# B&R Automation Studio project TD52 (part 27)

#### EleStartCyclic.st
```iecst
 (********************************************************************
EleStart		engine start/stop control: electrical starter equipment

This code is confidential and proprietary to the INNIO Company.
It may not be used in any form, or reproduced in any manner,
without the express written permission of the INNIO Company.
Copyright, INNIO Company, 2025

Customized modifications: -
------------------------

History:
-------
V01		10.07.1998 Pa			erstellt
V2.20.3	30.11.2007 LH			Ausspuren Starter bei Zahn auf Zahn
V2.30.0	16.01.2008 LH			Blockierung Modul angepasst für Insel nach Ablauf KU-Filter
 		30.01.2008 LH			Ansteuerung MEGA-Gasventile
 		02.04.2008 LH			1-maliges Absetzen von UW-EIN nach Kaltstart
V2.33.0	17.07.2008 lettenb.		sel_GlowIgnPrevent added
V2.34.0	22.10.2008 lettenb.		AT4_BLOCK added, block.ack.by starter temp.(op.message 3300)
								bs_15s_rel_oper added
		03.12.2008 lettenb.		ZM_GASV: M_GASV added
V2.50.0	28.01.2009 lettenb.		ZM_M_BLOCK: M_ST_VORW removed
			   	            	puff_mini removed
		06.04.2009 lett./gföll./plattner	Vorschmierzeit fix mit 60 = ersatz für TW_T85
								überbrückung T_VERZ_ANF bei notstrom(M_NANF)
V2.60.0	07.08.2009 lettenb.		udp_dmnd, udp_comm removed, ANF_NB added
								ssExtPwrSetP1, ssExtPwrSetP2, DI_ExtPwrSetP1, DI_ExtPwrSetP2 added
								custom.counter1-4 moved to c_amm
V3.10.0	19.01.2010 lettenb.		QUITT_TUEV reset pulse according EN ISO 13849-1 / 5.2.2
								(d.h. Ausgangsimpuls an UW_EIN erst wenn der RESET-Taster losgelassen wird)
V3.20.0	05.08.2010 lettenb.		ton_RESET_4 added reset counter for AT4_BLOCK after cool down
		15.09.2010 MM (BuR)  	STARTER_IgnST included
		30.09.2010 MM (BuR)  	GS_EIN replaced with GCB_ON
		30.09.2010 MM(BuR) 		NW20 deleted (GCB_ON --> GCB_ON)
		30.09.2010 MM(BuR) 		M_GSEIN replaced with GCB_ON
		21.10.2010 lettenb. 	AW_EXPSH, AW_EXPSB, B_P_SOLL, B_P_RED, AW_EXDSH, AW_EXDSB, B_N_SOLL
								sel.ext.power setpoint moved to task: p_limits
		05.11.2010 lettenb.		purgecycle added
		07.12.2010 lettenb.		BLOCK_EVU added, ZUEND: contact STARTER_IgnST changed
		14.02.2011 lettenb.		selection duration start puls time added
V3.90.0	29.10.2012 lettenb.		logic for manual start prozedure changed
V3.99.0	14.02.2013 lettenb.		IN_AG.bGasMix_Ref(M_GM_Ref) removed, not supported from MM gas mixer
V3.99   28.02.2013 pankajrodey	Generated for modular software with changes for V3.30
V3.99.1	20.01.2014 lettenb.		man.start time 30" added
V3.99.2	05.12.2013 zengerer		ADAPTIVE maximum start time 22" to 35" with rTiFactor_Cylinders AND rTiFactor_Cylinders FOR series 4 deflagration, new OUT: bRel_Gasvalve for MM op_state
V3.99.3	09.12.2013 zengerer		CleanUp
V3.99.4	02.01.2014 zengerer		prepared FOR PILOT ENGINES: save statistic data of 200 starts in task Perm_AG
V3.99.5	29.01.2014 zengerer		bGV_Start_ScaveBlock, MM2VIS.rN_EngStart (and others) optional reactivated
V3.99.6	19.03.2014 zengerer		entered Para.bVISA to prevent use of new adoptive start, if VISA reglementation is selected
V4.00.1 09.05.2014 lettenb.		xEngType.Type4: OUT_AG.tChargeOff_Dem.Do added, bugfix
V4.00.1 19.05.2014 Denk			xTON_StartErr Startzeit von 20s --> 12s
V4.00.2 30.05.2014 lettenb.		startup failure counter also for man.starts, bugfix + cleanup
V4.00.3 30.06.2014 lettenb.		xEngType.Type2 added, bugfix
V4.00.4 01.10.2014 lettenb.		bugfix startup failure in combination with EG_Scav(BR3,4)
		03.11.2014				start duration times BR3,6 corr., bugfix
V4.00.5	03.02.2015				920 added
		20.04.2015				xTP_StarterON: phantomstart resolved
V4.04.0	18.11.2016				xTON_DelayStart.PT, xTON_DelayManStart.PT: 6->0s start delay removed(fahringer)
		21.12.2016 Denk			Modification for WinMOD simulation
V4.05.0	07.08.2017 Messner		Starter battery voltage monitoring
		01.02.2018 lettenb.		tiStarterOFF; define value at plc startup(when xCTD_Start.CV=0), bugfix(1st start too long/perktold)
V4.05.1	14.02.2018 Weitzerr		move starter battery voltage monitoring to task AuxGnl
		19.09.2018 lettenb.		switching off battery charge for BR2+3 identical to BR4(HW solution not working), bu
V4.06.0	19.09.2018 Perktold,	integrated OUT_AG.iStartCount
V4.07.0	25.10.2018 Schmid		xTON_RESET_4: only triggered with IN_AG.bEng_SU_Man, bugfix
V4.10.0	28.01.2021 Schmid		interface for ChargeOff_Dem for starter battery test added
		29.01.2021 Schmid		manual start stop buttons from Opstate instead of VIS
V4.12.0 21.12.2022 Bacci		Starter battery monitoring parameters added: Para.rN_StarterMonTtT_LimLo and Para.tiStarterMonDuration. W9074 added
		20.01.2023 Zengerer		Type3 flush start time preparation optional with bOptType3AdoptiveStartEnab
V4.13.0	21.07.2023 Bacci		Type3 new starting procedure and adaptive first start attempt (bOptType3AdoptiveStartEnab deleted)
		20.11.2023 Bacci		Starter/s correct engagement monitoring added
V4.14.0	25.11.2024 Bacci		T6 Start procedure with purge start (2024-219)
V4.25.0	10.09.2025 Bacci	 	Include purge air calculation via SafetyPLC (2025-260)

Instructions for use:
--------------------
Outstandings:
------------
(*********************************************************************)

PROGRAM _CYCLIC

	(* Engine Type 9 - Return *)
	IF xEngType.Type9 THEN RETURN;
    END_IF;

	IF xEngType.Type6 THEN
		xR_TRIG_bParaSetupOk(CLK := IN_AG.tPB2MM.bParaSetupOk);
		IF xR_TRIG_bParaSetupOk.Q THEN
			rTi_ST_Active_zero := LIMIT(0, TIME_TO_REAL(Para.tiST_MaxDur_OverheatPrev)/1000 * (1 - (LIMIT(0.2, Para.rST_ReqOpTiAftCooldown, 1))), MAX(0,TIME_TO_REAL(Para.tiST_MaxDur_OverheatPrev)/1000));
		END_IF;
	ELSE
		rTi_ST_Active_zero := 0;
	END_IF;

	bAdoptiveStartEnab := (xEngType.Type4 OR xEngType.Type3) AND NOT Para.bVISA;

	IF xEngType.Type6 THEN							(* BR6 *)(* No longer used (2024-219) *)
		tiStarterON1 :=	 T#25s; 	(* = Total start time incl. flush cranking time at 1st start attempt in automatic *)
		tiStarterON2 :=	 T#20s;		(* = Total start time incl. flush cranking time at 2nd start attempt in automatic *)
		tiStarterON3 :=	 T#20s; 	(* = Total start time incl. flush cranking time at 3rd start attempt in automatic *)
		tiStartScav1 :=	 T#2s;		(* = flush cranking time wthout gas, for 1st start attempt *)
		tiStartScav2 :=	 T#2s;  	(* = flush cranking time wthout gas, for 2nd start attempt *)
		tiStartScav3 :=	 T#2s;  	(* = flush cranking time wthout gas, for 3rd start attempt *)
		tiStarterOFF1 := T#14s; 	(* = N.C. not in use *)
		tiStarterOFF2 := T#14s; 	(* = delay time until 2nd start attempt *)
		tiStarterOFF3 := T#14s; 	(* = delay time until 3rd start attempt *)
	ELSIF xEngType.Type4 AND NOT Para.bVISA THEN 	(* BR4 *)
		tiStarterON1 :=	 T#22s;		(* = Total start time incl. flush cranking time, base time for 1st start attempt- ADAPTIVE maximum time 22" (max.35" *)
		tiStarterON2 :=	 T#30s;		(* = Total start time incl. flush cranking time, for 2nd start attempt *)
		tiStarterON3 :=	 T#30s;		(* = Total start time incl. flush cranking time, for 3rd start attempt *)
		tiStartScav1 :=	 T#0s;		(* = flush cranking time wthout gas, for 1st start attempt- ADAPTIVE maximum time 22" to 35" *)
		tiStartScav2 :=	 T#10s;		(* = flush cranking time wthout gas, for 2nd start attempt *)
		tiStartScav3 :=	 T#10s;		(* = flush cranking time wthout gas, for 3rd start attempt *)
		tiStarterOFF1 := T#15s;		(* = n.c. *)
		tiStarterOFF2 := T#12s;		(* = delay time until 2nd start attempt *)
		tiStarterOFF3 := T#301s;	(* = delay time until 3rd start attempt *)
	ELSIF xEngType.Type3 AND NOT Para.bVISA THEN 		(* BR3 option with flush hardware *)
		tiStarterON1 :=	 T#34s;		(* = Total start time incl. flush cranking time, base time for 1st start attempt- ADAPTIVE maximum time 34" (max.40" *)
		tiStarterON2 :=	 T#30s;		(* = Total starg time incl. flush cranking time, time for 2nd start attempt *)
		tiStarterON3 :=	 T#30s;		(* = Total start time incl. flush cranking time, time for 3rd start attempt *)
		tiStartScav1 :=	 T#10s;		(* = flush cranking time wthout gas, for 1st start attempt- ADAPTIVE maximum time 22" to 35" *)
		tiStartScav2 :=	 T#10s;		(* = flush cranking time wthout gas, for 2nd start attempt *)
		tiStartScav3 :=	 T#10s;		(* = flush cranking time wthout gas, for 3rd start attempt *)
		tiStarterOFF1 := T#15s;		(* = n.c. *)
		tiStarterOFF2 := T#12s;		(* = delay time until 2nd start attempt *)
		tiStarterOFF3 := T#301s;	(* = delay time until 3rd start attempt *)
	ELSE											(* BR2,BR3 with standard hardware *)
		tiStarterON1 :=	 T#20s; 	(* = Total start time incl. flush cranking time, for 1st start attempt *)
		tiStarterON2 :=	 T#20s;		(* = Total start time incl. flush cranking time, for 2nd start attempt *)
		tiStarterON3 :=	 T#20s;		(* = Total start time incl. flush cranking time, for 3rd start attempt *)
		tiStartScav1 :=	 T#0s;		(* = flush cranking time wthout gas, for 1st start attempt *)
		tiStartScav2 :=	 T#0s;		(* = flush cranking time wthout gas, for 2nd start attempt *)
		tiStartScav3 :=	 T#0s;		(* = flush cranking time wthout gas, for 3rd start attempt *)
		tiStarterOFF1 := T#12s;		(* = n.c. *)
		tiStarterOFF2 := T#12s;		(* = delay time until 2nd start attempt *)
		tiStarterOFF3 := T#12s;		(* = delay time until 3rd start attempt *)
	END_IF;

	IF rTiFactor_Cylinders = 0 THEN	rTiFactor_Cylinders := 0.99; END_IF;
	IF rTiFactor_N_EngStart= 0 THEN	rTiFactor_N_EngStart:= 0.99; END_IF;

	(* start stop button info from Opstate *)
	bStart 	:= IN_AG.bStart;
	bStop 	:= IN_AG.bStop;

	(* -------------------------------------------------------------------------------------------------------------------------------------- *)
	(* New type 6 starting procedure *)

	(* ------------------------------------------------------------------------------------ *)
	(* EleStart cycle time *)
	RTInfo_CTR(enable := TRUE);
	tiCycleTime := UDINT_TO_TIME(RTInfo_CTR.cycle_time)/1000;		// time variable
	rCycleTime := UDINT_TO_REAL(RTInfo_CTR.cycle_time)/1000000;  	// real variable in seconds

	(* ------------------------------------------------------------------------------------ *)
	(* Set parameter 15074 "Minimum air volume required for system purge" based on parameter 11303 "exhaust gas scavenging active" and EPS demand *)
	IF xEngType.Type6 THEN
		IF NOT Para.bEGScav_Active THEN 				// Exhaust gas scavenging not active
			IF xEngType.Motortype = 612 THEN
				IF IN_AG.bEng_Dem_EPS THEN
					iVol_MinAirLim_SysPurge := 680;
				ELSE
					iVol_MinAirLim_SysPurge := MAX(680, Para.iVol_MinAir_SysPurge);
				END_IF;
			ELSIF xEngType.Motortype = 616 THEN
				IF IN_AG.bEng_Dem_EPS THEN
					iVol_MinAirLim_SysPurge := 750;
				ELSE
					iVol_MinAirLim_SysPurge := MAX(750, Para.iVol_MinAir_SysPurge);
				END_IF;
			ELSIF xEngType.Motortype = 620 THEN
				IF IN_AG.bEng_Dem_EPS THEN
					iVol_MinAirLim_SysPurge := 800;
				ELSE
					iVol_MinAirLim_SysPurge := MAX(800, Para.iVol_MinAir_SysPurge);
				END_IF;
			ELSIF xEngType.Motortype = 624 THEN
				IF IN_AG.bEng_Dem_EPS THEN
					iVol_MinAirLim_SysPurge := 1400;
				ELSE
					iVol_MinAirLim_SysPurge := MAX(1400, Para.iVol_MinAir_SysPurge);
				END_IF;
			END_IF;
		ELSIF Para.bEGScav_Active AND (IN_AG.bEng_Dem_EPS AND (NOT Para.bEGScav_ifAuxV_ok OR NOT IN_AG.tAuxV_Eng_ok.Di)) THEN 				// Exhaust gas scavenging active, but not executed during EPS
			IF xEngType.Motortype = 612 THEN
				iVol_MinAirLim_SysPurge := 680;
			ELSIF xEngType.Motortype = 616 THEN
				iVol_MinAirLim_SysPurge := 750;
			ELSIF xEngType.Motortype = 620 THEN
				iVol_MinAirLim_SysPurge := 800;
			ELSIF xEngType.Motortype = 624 THEN
				iVol_MinAirLim_SysPurge := 1400;
			END_IF;
		ELSE
			iVol_MinAirLim_SysPurge := 0;
		END_IF;
	ELSE
		iVol_MinAirLim_SysPurge := 0;
	END_IF;

	(* ------------------------------------------------------------------------------------ *)
	(* Volume flow through the engine *)
	IF xEngType.Type6 THEN
		rVol_CylDis :=	((UINT_TO_REAL(xEngType.Bore)/1000/2) ** 2 * brmPI * UINT_TO_REAL(xEngType.Stroke)/1000) * 1000; 								// single cylinder displacement [lt], //	Volume [lt]	:=	(( radius [m] ) ^ 2 * PI * ( stroke [m] ))*1000
		IF IN_AG.rN_EngAct > 50 THEN
			rVolFlow_RunEng := LIMIT(0, Para.rVolEff_CrkSpeed * rVol_CylDis * UINT_TO_REAL(xEngType.NumberOfCylinder) * IN_AG.rN_EngAct/120, 20000);	// volume flow through the engine REAL [lt/s]
		ELSE
			rVolFlow_RunEng := 0;
		END_IF;
		iVolFlow_RunEng := REAL_TO_UDINT(rVolFlow_RunEng);																								// volume flow through the engine UDINT [lt/s]
	ELSE
		rVol_CylDis := 0;
		rVolFlow_RunEng := 0;
		iVolFlow_RunEng := 0;
	END_IF;

	(* ------------------------------------------------------------------------------------ *)
	(* Volume of mixture calculation *)
	xTON_GVOpen_1s(IN:= IN_AG.bGV_On, PT:= T#1s);																								// gas valve open for more than 1 second

	IF xEngType.Type6 THEN
		//Fuel admition status
		IF xTON_GVOpen_1s.Q  THEN
			 rFuelAdm := 1;
		ELSE
			 rFuelAdm := (Para.rVolFlow_Marg - 1);
		END_IF;

		IF IN_AG.rN_EngAct = 0 OR OUT_AG.tEleStarter_Dem.Do THEN 																				// during engine standstill and during cranking phase
			rVol_Mx := LIMIT(0, rVol_Mx + rFuelAdm * rVolFlow_RunEng * rCycleTime, LIMIT(100, UDINT_TO_REAL(Para.iVol_TolUnbrtMxMax), 5000));
		ELSIF IN_AG.rN_EngAct <> 0 AND NOT IN_AG.bGV_On AND NOT OUT_AG.tEleStarter_Dem.Do  THEN													// during shut down phase
			rVol_Mx := LIMIT(0, rVol_Mx + rFuelAdm * rVolFlow_RunEng * rCycleTime, UDINT_TO_REAL(Para.iVol_PremxInSys));
		ELSIF M_DREHZ AND IN_AG.bGV_On THEN 																									// during engine operation
			rVol_Mx := UDINT_TO_REAL(Para.iVol_PremxInSys);
		END_IF;
	ELSE
		rFuelAdm := 0;
		rVol_Mx := 0;
	END_IF;

	(* ------------------------------------------------------------------------------------ *)
	(* Purge state identification *)
	IF xEngType.Type6 THEN
		(* Volume of purge air calculation *)
		IF IN_AG.bSafetyPLC_Active AND NOT Para.bEGScav_Active THEN 														//coming from safety PLC 	(* SAFETY PLC *)
			rVol_PurgeAir := IN_AG.rVol_PurgeAir_SafeOUT;																								(* SAFETY PLC *)
		ELSIF xTON_GVOpen_1s.Q OR bFail_PurgeCrk THEN																									(* SAFETY PLC *)
			rVol_PurgeAir := 0;
		ELSE
			rVol_PurgeAir := LIMIT(0, rVol_PurgeAir + rVolFlow_RunEng * (1 - Para.rVolFlow_Marg) * rCycleTime, 100000);		// volume of purge air REAL [lt]
		END_IF;
		iVol_PurgeAir := REAL_TO_UDINT(rVol_PurgeAir);																		// volume of purge air UDINT [lt]

		(* Purge state *)
		(* detect reset of emergancy operation demand  *)
		xF_TRIG_bEng_Dem_EPS(CLK := IN_AG.bEng_Dem_EPS);
		IF xF_TRIG_bEng_Dem_EPS.Q THEN
			bSt_Purge := FALSE;																								// set purge status to false after emergency operation demand reset
		END_IF;

		IF IN_AG.bSafetyPLC_Active AND NOT Para.bEGScav_Active THEN 														//coming from safety PLC 	(* SAFETY PLC *)
			bSt_Purge := IN_AG.bSafeOUT_Purge_OK;																										(* SAFETY PLC *)
		ELSIF xTON_GVOpen_1s.Q THEN 																													(* SAFETY PLC *)
			bSt_Purge := FALSE;
		ELSIF (rVol_PurgeAir >= UDINT_TO_REAL(iVol_MinAirLim_SysPurge)) THEN
			bSt_Purge := TRUE;
		END_IF;

		(* detect successful purge cranking cycle *)
		xR_TRIG_bSt_Purge(CLK := bSt_Purge);
	ELSE
		rVol_PurgeAir := 0;
		iVol_PurgeAir := 0;
		bSt_Purge := FALSE;
	END_IF;

	(* ------------------------------------------------------------------------------------ *)
	(* Starter temperature monitoring *)
	IF xEngType.Type6 THEN
		(* detect beginning of starter cool down phase *)
		xF_TRIG_bEleStarter_Dem(CLK := OUT_AG.tEleStarter_Dem.Do);
		IF xF_TRIG_bEleStarter_Dem.Q THEN
			rTi_ST_Active_zero := rTi_ST_Active;
			rTi_ST_Cooldown := 0;
		END_IF;

		(* Cumulated starting time calculation REAL [s] *)
		IF OUT_AG.tEleStarter_Dem.Do THEN
			rTi_ST_Active := LIMIT(0, rTi_ST_Active + Para.rST_Heatup_Fact * rCycleTime, MAX(0,TIME_TO_REAL(Para.tiST_MaxDur_OverheatPrev)/1000));																// Starter in use, heat up phase
		ELSE
			rTi_ST_Active := LIMIT(0, rTi_ST_Active_zero * EXP(-(rTi_ST_Cooldown / LIMIT(100, TIME_TO_REAL(Para.tiST_CooldownConst)/1000, 9000))), MAX(0,TIME_TO_REAL(Para.tiST_MaxDur_OverheatPrev)/1000));	// Starter not in use, cool down phase
			rTi_ST_Cooldown := rTi_ST_Cooldown + rCycleTime;
		END_IF;

		IF rTi_ST_Active < 1 AND NOT OUT_AG.tEleStarter_Dem.Do THEN 				// Rounding for small values
			rTi_ST_Active := 0;
			rTi_ST_Cooldown := 0;
			rTi_ST_Active_zero := 0;
		END_IF;

		(* Calculation of remaining starting time [s] *)
		rTi_ST_Res := TIME_TO_REAL(Para.tiST_MaxDur_OverheatPrev)/1000 - rTi_ST_Active;
		iTi_ST_Res := REAL_TO_INT(rTi_ST_Res);

		(* Calculation of starter temperature status *)
		xGR_MINR_bSt_STT (In:= rTi_ST_Res, Gw:= 0, Hy:= LIMIT(0, TIME_TO_REAL(Para.tiST_MaxDur_OverheatPrev)/1000 * (LIMIT(0.2, Para.rST_ReqOpTiAftCooldown, 1)), MAX(0,(TIME_TO_REAL(Para.tiST_MaxDur_OverheatPrev)/1000)-1)));
		bSt_STT := NOT xGR_MINR_bSt_STT.Q;
	ELSE
		rTi_ST_Active_zero := 0;
		rTi_ST_Cooldown := 0;
		rTi_ST_Active := 0;
		rTi_ST_Res := 0;
		iTi_ST_Res := 0;
		bSt_STT := FALSE;
	END_IF;

	//note:
	//		1.	the division by zero in the exponential calculation has been prevented using the boundaries limits decided for Para.tiST_CooldownConst
	//		2.	The upper limit of xGR_MINR_bSt_STT is used to be able to set the starter temperature status to true when Para.rST_ReqOpTiAftCooldown is 100%.
	//			In such situation, since rTi_ST_Res is never higher than TIME_TO_REAL(Para.tiST_MaxDur_OverheatPrev)/1000,  xGR_MINR_bSt_STT would never go to FALSE
	//			The cumulated starting time is forced to 0 when it´s value is < than 1s. The same trashold has been used also on the remining starting time.
	//			When rTi_ST_Res is > maximunm starting duration - 1s  the starter temperature status is set to TRUE (xGR_MINR_bSt_STT goes to false)

	(* ------------------------------------------------------------------------------------ *)
	(* Manual request for purge cranking cycle and start attempt *)
	IF xEngType.Type6 THEN
		bEng_SU_Man_Req := 		(bStart OR bEng_SU_Man_Req)
								AND		 bOMSS_Man
								AND 	 IN_AG.bEng_Dem_Man
								AND 	(IN_AG.bEng_SU_Man OR bSt_RelAuxOff_STT)								// retain during waiting time for starter release
								AND(NOT IN_AG.bBlocDelay_ManStart OR OUT_AG.bEng_Start OR bSt_RelAuxOff_STT)
								AND     (IN_AG.bScavFinished OR NOT IN_AG.bRel_ScavN2)
								AND NOT (xR_TRIG_bSt_Purge.Q AND xCTD_Start.CV <> xCTD_Start.PV)				// reset request when the purge done and first start
								AND NOT xF_TRIG_bSt_RelAuxOff_STT.Q												// reset request when release form starter temperature is given
								AND NOT bStop;
	ELSE
		bEng_SU_Man_Req := FALSE;
	END_IF;

	(* ------------------------------------------------------------------------------------ *)
	(* fast start readiness from purge status and starter temperature capability *)
	IF xEngType.Type6 THEN
		OUT_AG.bFS_Rdy_STT_StPurge := ((rTi_ST_Res >= TIME_TO_REAL(Para.tiST_MaxDur_OverheatPrev)/1000 * (LIMIT(0.2, Para.rST_ReqOpTiAftCooldown, 1))) AND bSt_Purge);		// enough starter temperature capability and purge ok
	ELSE
		OUT_AG.bFS_Rdy_STT_StPurge := FALSE;
	END_IF;

	(* ------------------------------------------------------------------------------------ *)
	(* demand to open inlet louvers before purge cranking cycle for fast start *)
	IF xEngType.Type6 THEN
		bFS_Req	:= bOMSS_Aut AND IN_AG.bEng_Rel AND Para.bFSPreL_Act AND IN_AG.bPermPreLube_Dem;
		OUT_AG.bInLouDemAG := (bFS_Req AND OUT_AG.bPreL_FS_EngStaRel AND NOT IN_AG.bEng_Bloc) AND NOT M_DREHZ AND NOT (bSt_Purge OR bStartAtt_Run);
	ELSE
		bFS_Req := FALSE;
		OUT_AG.bInLouDemAG := FALSE;
	END_IF;

	(* ------------------------------------------------------------------------------------ *)
	(* Purge cranking cycle *)
	IF xEngType.Type6 THEN
		// Request purge cranking cycle
		bReq_PurgeCrk := (IN_AG.bEng_Dem_Aut AND NOT M_DREHZ AND (IN_AG.bEng_SU_Aut OR (bSt_RelAuxOff_STT AND bPurgeCrk_Run)) AND NOT (bSt_Purge OR bStartAtt_Run)) OR								// request during automatic start attempt
						 (IN_AG.bEng_Dem_Man AND NOT M_DREHZ AND bEng_SU_Man_Req AND (IN_AG.bEng_SU_Man OR (bSt_RelAuxOff_STT AND bPurgeCrk_Run)) AND NOT (bSt_Purge OR bStartAtt_Run)) OR		 	// request during manual start attempt
						 ((bFS_Req AND OUT_AG.bPreL_FS_EngStaRel AND NOT IN_AG.bEng_Bloc) AND NOT M_DREHZ AND NOT (bSt_Purge OR bStartAtt_Run) AND IN_AG.bInLouRelVE);								// request from fast start

		IF bReq_PurgeCrk THEN														// function activation
			bPurgeCrk_Run := TRUE;													// purge cranking cycle running
			bReq_Rel_STT_PurgeCrk := TRUE; 											// starter temperature release function requested from purge cranking cycle
			bGV_Block_PurgeCrk := TRUE; 											// GV blocked during purge cranking cycle
			bDem_ST_PurgeCrk := NOT bSt_RelAuxOff_STT; 								// starter demand from purge cranking
			IF bSpeedMon_PurgeCrkStartAtt THEN 										// purge cranking speed monitoring
				IF NOT bFail_StartAtt THEN
					bFail_PurgeCrk := TRUE;											// A2376 purge cranking cycle unsuccessful
				END_IF;
				bPurgeCrk_Run := FALSE;
				bReq_Rel_STT_PurgeCrk := FALSE;
				bGV_Block_PurgeCrk := FALSE;
				bDem_ST_PurgeCrk := FALSE;
			END_IF;
		ELSIF xR_TRIG_bSt_Purge.Q AND bEleStarter_Dem_PurgeCrk THEN  				// purge cranking cycle completed.
			bSfl_PurgeCrk := TRUE;													// B9088 purge cranking cycle successful
			bPurgeCrk_Run := FALSE;
			bReq_Rel_STT_PurgeCrk := FALSE;
			//bGV_Block_PurgeCrk := FALSE;											// for one extra cycle the starter is kept on and GV blocked
			//bDem_ST_PurgeCrk := FALSE;
			IF bSpeedMon_PurgeCrkStartAtt THEN 										// purge cranking speed monitoring active also during this cycle
				bFail_PurgeCrk := TRUE;												// A2376 purge cranking cycle unsuccessful
				bSfl_PurgeCrk := FALSE;
			END_IF;
		ELSE
			bPurgeCrk_Run := FALSE;
			bReq_Rel_STT_PurgeCrk := FALSE;
			bGV_Block_PurgeCrk := FALSE;
			bDem_ST_PurgeCrk := FALSE;
			bSfl_PurgeCrk := FALSE;
		END_IF;

		(* messages *)
		xTP_bSfl_PurgeCrk(IN := bSfl_PurgeCrk, PT:= T#5s);
		bMsg9097_set	:= bPurgeCrk_Run AND iVol_MinAirLim_SysPurge <> 0; 				// 9097 "purge cranking cycle initiated "
		bMsg2376_T6_set	:= bFail_PurgeCrk; 												// 2376 for T6 "Purge cranking cycle unsuccessful"
		bMsg9088_T6_set	:= xTP_bSfl_PurgeCrk.Q AND iVol_MinAirLim_SysPurge <> 0; 		// 9088 for T6 "Purge cranking cycle successful" active for 5s
	ELSE
		bReq_PurgeCrk := FALSE;
		bSfl_PurgeCrk := FALSE;
		bPurgeCrk_Run := FALSE;
		bReq_Rel_STT_PurgeCrk := FALSE;
		bGV_Block_PurgeCrk := FALSE;
		bDem_ST_PurgeCrk := FALSE;
		bFail_PurgeCrk := FALSE;
		xTP_bSfl_PurgeCrk(IN := FALSE, PT:= T#0s);
		bMsg9097_set := FALSE;
		bMsg2376_T6_set := FALSE;
		bMsg9088_T6_set := FALSE;
	END_IF;

	(* ------------------------------------------------------------------------------------ *)
	(* Start attempt*)
	IF xEngType.Type6 THEN
		// Request starter temperature release before engine start attempt
		xR_TRIG_bReq_Rel_STT_StartAtt(CLK := ((IN_AG.bEng_SU_Aut AND NOT M_DREHZ AND bSt_Purge AND NOT xCTD_Start.Q) OR
									 		  (IN_AG.bEng_SU_Man AND bEng_SU_Man_Req AND NOT M_DREHZ AND bSt_Purge AND NOT xCTD_Start.Q)));

		IF xR_TRIG_bReq_Rel_STT_StartAtt.Q THEN
			bRel_STT_StartAtt := FALSE;
		END_IF;

		bReq_StartAtt := (IN_AG.bEng_Dem_Aut AND NOT M_DREHZ AND (IN_AG.bEng_SU_Aut AND (bSt_Purge OR bStartAtt_Run)) AND bRel_STT_StartAtt AND NOT xCTD_Start.Q) OR
						 (IN_AG.bEng_Dem_Man AND NOT M_DREHZ AND bEng_SU_Man_Req AND (IN_AG.bEng_SU_Man AND (bSt_Purge OR bStartAtt_Run)) AND bRel_STT_StartAtt AND NOT xCTD_Start.Q);

		xR_TRIG_bReq_StartAtt(CLK := bReq_StartAtt);
		(* detect engine demanded and purge cranking cycle done *)
		IF xR_TRIG_bReq_StartAtt.Q THEN
			rTiStartAttDur := 0;
			rVol_Mx := 0;
		END_IF;

		IF bReq_StartAtt THEN
			bStartAtt_Run := TRUE;											// start attempt running
			bDem_ST_StartAtt := TRUE; 										// starter demand from start attempt
			IF OUT_AG.tEleStarter_Dem.Do THEN
				rTiStartAttDur := rTiStartAttDur + rCycleTime;				// start attempt duration when starter demanded
			END_IF;
			IF rTiStartAttDur > 30 OR rVol_Mx >= LIMIT(100, UDINT_TO_REAL(Para.iVol_TolUnbrtMxMax), 5000) OR bSpeedMon_PurgeCrkStartAtt THEN		// start attempt duration, volume of mixture, speed monitoring
				bStartAtt_Run := FALSE;
				//bDem_ST_StartAtt := FALSE;
					IF bSpeedMon_PurgeCrkStartAtt THEN
						bDem_ST_StartAtt := FALSE;
						bFail_StartAtt := TRUE;
					END_IF;
			END_IF;
		ELSE
			bStartAtt_Run := FALSE;
			bDem_ST_StartAtt := FALSE;
		END_IF;

		bMsg2382_set	:= bFail_StartAtt; 									// A2382 for T6 "Start attempt failed minimum speed"
	ELSE
		bRel_STT_StartAtt := FALSE;
		bReq_StartAtt := FALSE;
		rTiStartAttDur := 0;
		bStartAtt_Run := FALSE;
		bDem_ST_StartAtt := FALSE;
		bFail_StartAtt := FALSE;
		bMsg2382_set := FALSE;
	END_IF;

	(* ------------------------------------------------------------------------------------ *)
	(* Waiting for starter temperature release / pause of pre-lubrication pump *)
	IF xEngType.Type6 THEN
		rTi_ST_Active_AftCooldown := LIMIT(1, TIME_TO_REAL(Para.tiST_MaxDur_OverheatPrev)/1000 * (1-(LIMIT(0.2, Para.rST_ReqOpTiAftCooldown, 1))), MAX(1, TIME_TO_REAL(Para.tiST_MaxDur_OverheatPrev)/1000)); 		// cumulated starting time after cooldown phase [s]

		// Detect exhaust scavenging procedure needed after purge cycle
		xF_TRIG_GVopen_bEGScavAct(CLK:= IN_AG.bGV_On AND Para.bEGScav_Active AND
										(NOT IN_AG.bEng_Dem_EPS OR (Para.bEGScav_ifAuxV_ok AND IN_AG.tAuxV_Eng_ok.Di)));

		// Request release from starter temperature
		bReq_Rel_STT := ((xR_TRIG_bEng_Dem_Aut.Q OR (IN_AG.bEng_Dem_Aut AND bSt_RelAuxOff_STT AND NOT M_DREHZ)) OR																		// Check for starter temperature release when engine demanded in automatic and retain function till the end of it
						(bReq_Rel_STT_PurgeCrk) OR 																																		// Check for starter temperature release during purge cranking cycle
						((xR_TRIG_bReq_Rel_STT_StartAtt.Q AND NOT xF_TRIG_GVopen_bEGScavAct.Q) OR ((IN_AG.bEng_Dem_Aut OR IN_AG.bEng_Dem_Man) AND bSt_RelAuxOff_STT AND NOT M_DREHZ)));	// Check for starter temperature release before automatic or manual start attempt and retain function till the end of it

		IF bReq_Rel_STT  THEN 																								// function activation
			bRel_STT_Ena := TRUE;																							// function enabled
			IF (bSt_STT AND (NOT bSt_Purge OR (bSt_Purge AND rTi_ST_Res >= (TIME_TO_REAL(Para.tiST_MaxDur_OverheatPrev)/1000 * (LIMIT(0.2, Para.rST_ReqOpTiAftCooldown, 1))))) OR IN_AG.bEng_Dem_EPS) THEN
				bPreLubeOff_STT := FALSE;																					// signal to stop prelubrication (when true) due to starter overheat
				bSt_RelAuxOff_STT := FALSE; 																				// signal to deactivate the starter (when true) due to starter overheat
				bRel_STT_StartAtt := TRUE;
			ELSE
				IF IN_AG.rN_EngAct = 0 THEN
					bPreLubeOff_STT := TRUE;
				END_IF;
				bSt_RelAuxOff_STT := TRUE;
				IF NOT OUT_AG.tEleStarter_Dem.Do THEN
					rTi_ST_UntRelDur := (-((LIMIT(100, TIME_TO_REAL(Para.tiST_CooldownConst)/1000, 9000)) * LN(rTi_ST_Active_AftCooldown / LIMIT (1, rTi_ST_Active_zero, MAX(1, TIME_TO_REAL(Para.tiST_MaxDur_OverheatPrev)/1000))))) - rTi_ST_Cooldown;		// duration in seconds till the release of the starter due to temperature
				END_IF;
			END_IF;
		ELSE
			bRel_STT_Ena := FALSE;
			bPreLubeOff_STT := FALSE;
			bSt_RelAuxOff_STT := FALSE;
		END_IF;

		(* messages *)
		(* 9096 "Starter overheated" *)
		xTON_bSt_RelAuxOff_STT(IN:= bSt_RelAuxOff_STT, PT:= T#1s);		//1s delay before setting the message 9096. to be sure that the additional information get stored with the operating message

		bMsg9096_enable := bRel_STT_Ena OR xTP_bMsg9096_set_retain.Q;
		bMsg9096_set := xTON_bSt_RelAuxOff_STT.Q OR xTP_bMsg9096_set_retain.Q;
		bMsg9096_iTi_ST_UntRelDur := REAL_TO_DINT(rTi_ST_UntRelDur);

		(* "Start up failure" when starter waiting time is higher than 600s *)
		bStartErr_ST_UntRelDur_High	:= bRel_STT_Ena AND bSt_Purge AND xTON_bSt_RelAuxOff_STT.Q AND rTi_ST_UntRelDur > 600;

		(* retain 9096 set for 20s when start up failure is activated *)
		xTP_bMsg9096_set_retain(IN:= bStartErr_ST_UntRelDur_High, PT:= T#20s);

		(* detect when the starter temperature release is given *)
		xF_TRIG_bSt_RelAuxOff_STT(CLK := bSt_RelAuxOff_STT);

		(* Starter request during start attempt *)
		bEleStarter_Dem_StartAtt := bDem_ST_StartAtt;

		(* Starter request during purge cranking cycle and released form strater temperature monitoring *)
		bEleStarter_Dem_PurgeCrk := bDem_ST_PurgeCrk AND NOT bSt_RelAuxOff_STT;

		(* Starter temperature release off for op_state and CBM *)
		OUT_AG.bSt_RelAuxOff_STT_op	:= bSt_RelAuxOff_STT;
	ELSE
		rTi_ST_Active_AftCooldown := 1;
		bReq_Rel_STT := FALSE;
		bRel_STT_Ena := FALSE;
		bPreLubeOff_STT := FALSE;
		bSt_RelAuxOff_STT := FALSE;
		bRel_STT_StartAtt := FALSE;
		rTi_ST_UntRelDur := 0;
		bMsg9096_enable := FALSE;
		bMsg9096_set := FALSE;
		bMsg9096_iTi_ST_UntRelDur := FALSE;
		bStartErr_ST_UntRelDur_High := FALSE;
		bEleStarter_Dem_StartAtt := FALSE;
		bEleStarter_Dem_PurgeCrk := FALSE;
		OUT_AG.bSt_RelAuxOff_STT_op := FALSE;
	END_IF;

	//note:
	//		1.	To avoid problem logaritm formula:
	//			The division by zero is avoided limiting cumulated starting time to a minimum value of 1s
	//			The wanted active starting time after cool down time (rTi_ST_Active_AftCooldown) has also been lower limited to 1s to avoid that the logaritm goes to infinite when Para.rST_ReqOpTiAftCooldown is set to 100%

	(* ------------------------------------------------------------------------------------ *)
	(* -------------------------------------------------------------------------------------------------------------------------------------- *)

	(* delay automatic start *)
	xTON_DelayStart(IN:= IN_AG.bEng_SU_Aut AND NOT bOMSS_Man, PT:= T#0s);
	OUT_AG.bEngAutStartDelay := xTON_DelayStart.Q;

	(* manual start *)
	ZM_HSTART	:= (bStart OR ZM_HSTART)
			AND		bOMSS_Man
			AND 	IN_AG.bEng_SU_Man
			AND(NOT IN_AG.bBlocDelay_ManStart OR     OUT_AG.bEng_Start)
			AND    (IN_AG.bScavFinished       OR NOT IN_AG.bRel_ScavN2)
			AND NOT xTP_StarterOFF.Q
			AND NOT bStop;

	(* delay manual start *)
	xTON_DelayManStart(IN:= ZM_HSTART AND bOMSS_Man, PT:= T#0s);

	(* set starter pulse ON-time *)
	IF IN_AG.bEng_SU_Man THEN		(*active only for auto starts*)
		tiStarterON_Base		:=	T#30s;  (* manual start time 30" *)
		tiStartScav				:=	T#0s;
		tiStarterOFF			:=	T#12s;
		bCalcAdaptiveStartTime	:=	FALSE;
	ELSE
		CASE xCTD_Start.CV OF
			3: 	tiStarterON_Base := tiStarterON1;
				tiStartScav      := tiStartScav1;
				tiStarterOFF     := tiStarterOFF1;
				IF bAdoptiveStartEnab (*xEngType.Type4 AND NOT Para.bVISA AND bDebugStartActive*) THEN	// activation for series 4 engines and marked as pilot activation bit
					bCalcAdaptiveStartTime := TRUE;
				END_IF;
			2: 	tiStarterON_Base := tiStarterON2;
				tiStartScav      := tiStartScav2;
				tiStarterOFF     := tiStarterOFF2;
				bCalcAdaptiveStartTime := FALSE;
			1: 	tiStarterON_Base := tiStarterON3;
				tiStartScav      := tiStartScav3;
				tiStarterOFF     := tiStarterOFF3;
				bCalcAdaptiveStartTime := FALSE;
			ELSE
				tiStarterON_Base := T#20s10ms;			(*check!*)
				tiStarterOFF     := tiStarterOFF1;
				bCalcAdaptiveStartTime := FALSE;
		END_CASE;
	END_IF;

	(* ------------------------------------------------------------------------------------ *)
	(* adopt starter puls ON-time for 1st. automatic start (Type4) *)
	bDebugStartActive := (IN_AG.rN_EngAct > 60);			(*detect turning starter *)

	xRT_bDebugStartActive(CLK:= bDebugStartActive);			(*detect turning starter delay*)
	IF xRT_bDebugStartActive.Q THEN
		bDebugStartActive_Delay := xTON_H_STRT.ET;
	END_IF;

	xTON_StarterMeas2(IN:=bDebugStartActive, PT:= T#5s);
	bDebugTON_StarterMeas2 := xTON_StarterMeas2.Q;

	xTP_StarterMeas(IN:= xTON_StarterMeas2.Q, PT:= T#1s);	(*timer for 1 sec start speed measurement *)
	bTriggerStarterMeas := xTP_StarterMeas.Q;
	xF_TRIG_StarterMeas(CLK := xTP_StarterMeas.Q);			(*trigger moment for calculation*)

	IF bCalcAdaptiveStartTime AND OUT_AG.bEng_Start THEN
		(* measure 1 sec speed average for calculation *)
		IF xTP_StarterMeas.Q  THEN
			rN_EngStartAvg := (rN_EngStartAvg * rCnt_EngStartAvg) +  IN_AG.rN_EngAct;  	(* speed average *)
			rCnt_EngStartAvg := rCnt_EngStartAvg + 1;
			IF rCnt_EngStartAvg > 0 THEN rN_EngStartAvg := rN_EngStartAvg / rCnt_EngStartAvg ; END_IF;
		ELSE
			rCnt_EngStartAvg := 0;
		END_IF;

		(* factor for cylinder number ADAPTIVE maximum time" *)
		LCRScal_Cylinders(x := xEngType.NumberOfCylinder , x1 := 12, y1 := 1.27, x2 := 20, y2 := 1);
		rTiFactor_Cylinders := LCRScal_Cylinders.y ;

	ELSE
		ti_EngStart_Max := 	xTP_StarterON.PT ;
	END_IF;

	IF bCalcAdaptiveStartTime AND xF_TRIG_StarterMeas.Q THEN
		MM2VIS.rN_EngStart :=	rN_EngStartAvg;		(*speed, for VIS*)
		rN_EngStart :=			rN_EngStartAvg;		(*speed, for VIS*)

		LCRScal_N_EngStart(x := rN_EngStartAvg, x1 := 130, y1 := 1.22, x2 := 170, y2 := 1);
		rTiFactor_N_EngStart :=  LIMIT(1.0, LCRScal_N_EngStart.y, 1.22);

		IF xEngType.Type3 THEN
			rStarterON_Max :=  LIMIT(24000, (TIME_TO_REAL(tiStarterON_Base - tiStartScav) * rTiFactor_Cylinders * rTiFactor_N_EngStart),38000) ;	(* 1. start ADAPTIVE maximum time 24" to 38" *)
			tiStarterON_Max := REAL_TO_TIME(rStarterON_Max) + tiStartScav;
		ELSE
			rStarterON_Max :=  LIMIT(20000, (TIME_TO_REAL(tiStarterON_Base) * rTiFactor_Cylinders * rTiFactor_N_EngStart),35000) ;	(* 1. start ADAPTIVE maximum time 20" to 35" *)
			tiStarterON_Max := REAL_TO_TIME(rStarterON_Max);
		END_IF;

		xTP_StarterON.PT := tiStarterON_Base ;
		IF  (tiStarterON_Max - xTON_StarterMeas2.PT - xTP_StarterMeas.PT) > T#0s THEN
			xTP_StarterON_Extended.PT := tiStarterON_Max - xTON_StarterMeas2.PT - xTP_StarterMeas.PT - bDebugStartActive_Delay;		(* 1. start additional maximum time 22" to 35" (type 4) 24" to 38" (type 3) *)
			xTP_StarterON_Extended.IN := bCalcAdaptiveStartTime;	 (*trigger the extended start time once*)
		ELSE
			xTP_StarterON_Extended.PT := 0;
		END_IF;
		MM2VIS.rTi_EngStart_Max := TIME_TO_REAL(tiStarterON_Max);		(*for VIS*)		//OPTIONAL 2014; no visu display
		ti_EngStart_Max := 						tiStarterON_Max ;
	ELSE
		IF NOT xTP_StarterON_Extended.Q THEN
			xTP_StarterON_Extended.PT := 0;
		END_IF;
	END_IF;
	xTP_StarterON_Extended();				(*timer FUB call for additional start time*)
	xTP_StarterON_Extended.IN := FALSE;

	IF T_H_STRT THEN  						(*limit xTP_StarterON_Extended to max start time*)
		xTP_StarterON_Extended.PT := 0;
	END_IF;

	xTP_StarterON.PT := tiStarterON_Base + xTON_ChargeOff.PT;		(*adding the charge off delay to correct the starter time Perktold 17.03.2023*);

	(* ------------------------------------------------------------------------------------ *)
	(* starter pulse ON-time *)
	T7_TEMP1 := (IN_AG.bEng_Dem_EPS AND NOT IN_AG.bOnly_Island) OR OUT_AG.bEngAutStartDelay;

	IF NOT IN_AG.bEng_Dem_EPS AND NOT ZM_HSTART AND NOT IN_AG.bEng_SU_Aut THEN (* reset timer *)
		xTP_StarterON(IN:= FALSE, PT:= T#0s);
	ELSIF IN_AG.bEng_SU_Man THEN
		xTP_StarterON(IN:= xTON_DelayManStart.Q AND NOT xTP_StarterOFF.Q);
	ELSIF IN_AG.bEng_SU_Aut THEN
		xTP_StarterON(IN:= T7_TEMP1             AND NOT xTP_StarterOFF.Q);
	ELSE
		xTP_StarterON(IN:= FALSE, PT:= T#0s);
	END_IF;
	bTP_StarterON := xTP_StarterON.Q
				OR	(xTP_StarterON_Extended.Q AND bCalcAdaptiveStartTime AND bAdoptiveStartEnab) ;  (*NEW 2014*)

	(* starter puls OFF-time *)
	xTP_StarterOFF(IN:= NOT bTP_StarterON, PT:= tiStarterOFF);

	(* ------------------------------------------------------------------------------------ *)
	//monitoring start ton_RESET_4 time for starter cool down = same time as for OUT_AG.bLockAckStarter
	xR_TRIG_Reset1(CLK:= IN_AG.tEng_Run.Do);
	xR_TRIG_Reset2(CLK:= IN_AG.bEng_Dem_Man_SUpF);
	xR_TRIG_Reset3(CLK:= IN_AG.bEng_Dem_Aut_SUpF);

	(* start counter reset after long pause between start attempts in manual mode *)
	xTON_Reset4(IN := NOT OUT_AG.bEng_Start AND IN_AG.bEng_SU_Man, PT:= T#300s);	(* serie *)
	xR_TRIG_Reset4(CLK:= xTON_Reset4.Q);

	RESET := xR_TRIG_Reset1.Q OR xR_TRIG_Reset2.Q OR xR_TRIG_Reset3.Q OR xR_TRIG_Reset4.Q;

	(*---------------------------------------------------------------------------------------------*)
	xF_TRIG_Start(CLK:= (bTP_StarterON AND NOT xEngType.Type6) OR (bStartAtt_Run AND xEngType.Type6));

	(* start counter *)
	xCTD_Start(CD:= xF_TRIG_Start.Q, LOAD:= RESET, PV:= 3);	//serie, xF_TRIG_Start war xR_TRIG_Start ?
	OUT_AG.iStartCount	:= LIMIT(1, xCTD_Start.PV - xCTD_Start.CV + 1, xCTD_Start.PV);  //Number of Start for OpState

	(* man + auto start error *)
	xTON_StartErr(IN:= xCTD_Start.Q AND NOT M_DREHZ AND(IN_AG.bEng_Dem_Aut_SUpF OR IN_AG.bEng_Dem_Man_SUpF) AND (bSt_Purge OR NOT xEngType.Type6), PT:= T#12s); (* delay = min.starter off interval time *)
	bStartErr := xTON_StartErr.Q;

	(*---------------------------------------------------------------------------------------------*)
	//blocking acknowledgement by starter temperature (op.message 3300)
	IF (xEngType.Type3 OR xEngType.Type4 OR xEngType.Type2) THEN
		xR_TRIG_AutoStartErr(CLK:= bStartErr);
		xTOF_LockAckStarter(IN:= xR_TRIG_AutoStartErr.Q, PT:= T#5m);
		IF IN_AG.bEng_Dem_EPS THEN
			xTOF_LockAckStarter(IN:= FALSE, PT:= T#0m);
		END_IF;
		OUT_AG.bLockAckStarter := xTOF_LockAckStarter.Q;
	ELSIF (xEngType.Type6) THEN
		OUT_AG.bLockAckStarter := FALSE;
	END_IF;

	(*---------------------------------------------------------------------------------------------*)
	(* start *)
	ZM_STRT   := IN_AG.bEng_Rel AND NOT M_DREHZ AND OUT_AG.bRelEngOp_Aux;

	IF xEngType.Type2 OR xEngType.Type3 OR xEngType.Type4 THEN
//		M_STRT_TEMP1 := NOT IN_AG.bBlocDelay_ManStart OR OUT_AG.bEng_Start;

		(* start release from EG scavening *)
//		M_STRT_TEMP2 := IN_AG.bScavFinished OR NOT IN_AG.bRel_ScavN2;

		(* manual start *)
		M_STRT_TEMP3 := ZM_STRT AND bTP_StarterON AND ZM_HSTART AND NOT T_H_STRT ;

		(* automatic start *)
		M_STRT_TEMP4 := ZM_STRT AND bTP_StarterON AND (OUT_AG.bEngAutStartDelay OR IN_AG.bEng_Dem_EPS) AND NOT T_H_STRT ;	(*neu: max mit T_H_STRT*)

		(* start demand from N2_scavenging *)
		M_STRT_TEMP6 := IN_AG.bN2_ScavCoStarterOn AND NOT M_DREHZ AND IN_AG.bRel_ScavN2;

		(* start demand from ignition selftest *)
		M_STRT_TEMP7 := IN_AG.b_ST_DemIgn         AND NOT M_DREHZ;

		bChargeOff_EngStart			:=	M_STRT_TEMP3 	(* man  start *)
									OR	M_STRT_TEMP4	(* auto start *)
									OR	M_STRT_TEMP6	(* N2_scavenging *)
									OR	M_STRT_TEMP7;	(* ignition selftest *)
		OUT_AG.tChargeOff_Dem.Do	:=	bChargeOff_EngStart OR bStarterBat_Disconnect;

		// Delay start relay after switching off battery charge
		xTON_ChargeOff(IN := bChargeOff_EngStart, PT := T#300ms);

		OUT_AG.bEng_Start         := xTON_ChargeOff.Q;

		xRT_EngStart(CLK:= OUT_AG.bEng_Start);						(* begin of start *)
		xFT_EngStart(CLK:= OUT_AG.bEng_Start);						(* end of start *)
		IF xRT_EngStart.Q AND b_EleStarter_EngageFail THEN
			b_EleStarter_EngageFail	:= FALSE;
			bEleStarterFail_Num[1]	:= FALSE;
			bEleStarterFail_Num[2]	:= FALSE;
			bEleStarterFail_Num[3]	:= FALSE;
		END_IF;

		OUT_AG.tEleStarter_Dem.Do := xTON_ChargeOff.Q AND NOT STP_STRT AND NOT b_EleStarter_EngageFail;

	ELSIF xEngType.Type6 THEN
		xTON_Nospeed15s(IN := IN_AG.rN_EngAct = 0.0, PT:= T#15s);
		bRel_Nospeed := (xTON_Nospeed15s.Q OR OUT_AG.bEng_Start);

		M_STRT_TEMP4 := (bEleStarter_Dem_PurgeCrk OR bEleStarter_Dem_StartAtt) AND (bRel_Nospeed);
		M_STRT_TEMP5 := M_STRT_TEMP4 AND (ZM_STRT OR OUT_AG.bPreL_FS_EngStaRel); 									// during purge while fast start preparation the aux release for engine operation won´t be there, used permanent prelubrication feedback
		M_STRT_TEMP6 := IN_AG.bN2_ScavCoStarterOn AND NOT M_DREHZ AND IN_AG.bRel_ScavN2;
		M_STRT_TEMP7 := IN_AG.b_ST_DemIgn AND NOT M_DREHZ;

		bChargeOff_EngStart			:= M_STRT_TEMP5 OR M_STRT_TEMP6 OR M_STRT_TEMP7;

		OUT_AG.tChargeOff_Dem.Do	:= bChargeOff_EngStart OR bStarterBat_Disconnect;

		// Delay start relay after switching off battery charge
		xTON_ChargeOff(IN := bChargeOff_EngStart, PT:= T#300ms);

		OUT_AG.bEng_Start         := xTON_ChargeOff.Q;

		xRT_EngStart(CLK:= OUT_AG.bEng_Start);						(* begin of start *)
		xFT_EngStart(CLK:= OUT_AG.bEng_Start);						(* end of start *)
		IF xRT_EngStart.Q AND b_EleStarter_EngageFail THEN
			b_EleStarter_EngageFail := FALSE;
			bEleStarterFail_Num[1]	:= FALSE;
			bEleStarterFail_Num[2]	:= FALSE;
			bEleStarterFail_Num[3]	:= FALSE;
		END_IF;

		OUT_AG.tEleStarter_Dem.Do := xTON_ChargeOff.Q AND NOT STP_STRT AND NOT b_EleStarter_EngageFail;

		(* starter demand during purge cranking cycle *)
		OUT_AG.bEleStarter_Dem_PurgeCrkCyl := OUT_AG.tEleStarter_Dem.Do AND bEleStarter_Dem_PurgeCrk;

		(* starer demanded during purge cranking cycle for fast start preparation *)
		IF OUT_AG.tEleStarter_Dem.Do AND bEleStarter_Dem_PurgeCrk AND bFS_Req AND NOT IN_AG.bEng_Dem THEN
			OUT_AG.bEleStarter_Dem_PurgeCrkCylFS := TRUE;
		ELSIF OUT_AG.bEleStarter_Dem_PurgeCrkCylFS AND (IN_AG.rN_EngAct = 0.0 OR IN_AG.bEng_Dem) THEN
			OUT_AG.bEleStarter_Dem_PurgeCrkCylFS := FALSE;
		END_IF;
	END_IF;

	// Starter/s correct engagement monitoring
	xTON_EleStarter_Mon	(IN := OUT_AG.tEleStarter_Dem.Do, PT := Para.tiStarterFunDuration);			(* starter/s correct engagement monitoring trigger *)
	xTP_EleStarter_Mon	(IN	:= xTON_EleStarter_Mon.Q, PT:= T#300ms);								(* 300ms timer for voltage measurement *)
	xFT_EleStarter_Mon	(CLK:= xTP_EleStarter_Mon.Q);												(* correct engagement monitoring evaluation instant *)

	IF OUT_AG.tEleStarter_Dem.Do AND xTP_EleStarter_Mon.Q THEN
		rU_EleStarterAvg1 := (rU_EleStarterAvg1 * rCnt_EleStarterAvg) +  IN_AG.tU_Starter_engage1.Ai;
		rU_EleStarterAvg2 := (rU_EleStarterAvg2 * rCnt_EleStarterAvg) +  IN_AG.tU_Starter_engage2.Ai;
		rU_EleStarterAvg3 := (rU_EleStarterAvg3 * rCnt_EleStarterAvg) +  IN_AG.tU_Starter_engage3.Ai;

		rCnt_EleStarterAvg := rCnt_EleStarterAvg + 1;

		IF rCnt_EleStarterAvg > 0 THEN
			rU_EleStarterAvg1 := rU_EleStarterAvg1 / rCnt_EleStarterAvg;    (* starter 1 terminal 45 average voltage *)
			rU_EleStarterAvg2 := rU_EleStarterAvg2 / rCnt_EleStarterAvg;  	(* starter 2 terminal 45 average voltage *)
			rU_EleStarterAvg3 := rU_EleStarterAvg3 / rCnt_EleStarterAvg;   	(* starter 3 terminal 45 average voltage *)
		END_IF;
	ELSE
		rCnt_EleStarterAvg := 0;
	END_IF;

	IF Para.rU_StarterMon_LimLo <> 0 THEN 																								(* active monitoring if parameter different than zero *)
		IF xFT_EleStarter_Mon.Q AND OUT_AG.tEleStarter_Dem.Do THEN 																		(* measurement completed and starter demand still ON *)
			IF (IN_AG.tU_Starter_engage1.GoodQual AND NOT MM2VIS.bMsg2377 AND rU_EleStarterAvg1 < Para.rU_StarterMon_LimLo) THEN		(* average voltage too low *)
				b_EleStarter_EngageFail	:= TRUE;																						(* starter motor did not engage*)
				bEleStarterFail_Num[1]	:= TRUE;
			END_IF;
			IF (IN_AG.tU_Starter_engage2.GoodQual AND NOT MM2VIS.bMsg2378 AND rU_EleStarterAvg2 < Para.rU_StarterMon_LimLo) THEN
				b_EleStarter_EngageFail := TRUE;
				bEleStarterFail_Num[2]	:= TRUE;
			END_IF;
			IF (IN_AG.tU_Starter_engage3.GoodQual AND NOT MM2VIS.bMsg2379 AND rU_EleStarterAvg3 < Para.rU_StarterMon_LimLo) THEN
				b_EleStarter_EngageFail := TRUE;
				bEleStarterFail_Num[3]	:= TRUE;
			END_IF;
		END_IF;
	ELSE
		b_EleStarter_EngageFail	:= FALSE;
		bEleStarterFail_Num[1]	:= FALSE;
		bEleStarterFail_Num[2]	:= FALSE;
		bEleStarterFail_Num[3]	:= FALSE;
	END_IF;

	// trip starter if tooth to tooth
	xTON_ZAZ(IN := OUT_AG.bEng_Start AND (IN_AG.rN_EngAct < Para.rN_StarterMonTtT_LimLo), PT := Para.tiStarterMonDuration);
	STP_STRT    := xTON_ZAZ.Q;

	(* Speed monioring during purge cranking cycle and start attempt *)
	xGR_MAXR_SpeedMon(In := IN_AG.rN_EngAct, Gw:= 62.0, Hy := 2.0);	// detect speed drop below 60 rpm
	xF_TRIG_SpeedMon(CLK:= xGR_MAXR_SpeedMon.Q);

	IF xEngType.Type6 THEN
		bSpeedMon_PurgeCrkStartAtt :=	((OUT_AG.bEng_Start AND (bEleStarter_Dem_PurgeCrk OR bEleStarter_Dem_StartAtt)) AND 		// engine start and purge cranking or start attempt running
										(xTON_ZAZ.Q OR 							// tooth to tooth detection
										xF_TRIG_SpeedMon.Q) OR					// speed drops below 60rpm
										bFail_PurgeCrk OR bFail_StartAtt); 		// retain when failed purge cycle or start attempt
	ELSE
		bSpeedMon_PurgeCrkStartAtt := FALSE;
	END_IF;

	(*---------------------------------------------------------------------------------------------*)
	(* maximum start time *)
	IF xEngType.Type2 THEN
		xTON_H_STRT(IN:= OUT_AG.bEng_Start, PT:= T#30s);
	ELSIF xEngType.Type3 THEN
		IF xEngType.NumberOfCylinder = 12 THEN
			xTON_H_STRT(IN:= OUT_AG.bEng_Start, PT:= T#48s);
		ELSIF xEngType.NumberOfCylinder = 16 THEN
			xTON_H_STRT(IN:= OUT_AG.bEng_Start, PT:= T#44s);
		ELSIF xEngType.NumberOfCylinder = 20 THEN
			xTON_H_STRT(IN:= OUT_AG.bEng_Start, PT:= T#40s);
		ELSE
			xTON_H_STRT(IN:= OUT_AG.bEng_Start, PT:= T#40s);
		END_IF;
	ELSIF xEngType.Type4 THEN
		xTON_H_STRT(IN:= OUT_AG.bEng_Start, PT:= T#35s);
	ELSIF xEngType.Type6 THEN
		xTON_H_STRT(IN:= OUT_AG.bEng_Start, PT:= T#30s);
	END_IF;
	T_H_STRT := xTON_H_STRT.Q;

	(*---------------------------------------------------------------------------------------------*)
	(* start scavenging time with ignition on (only type 3 and 6)*)
	IF xEngType.Type3 OR xEngType.Type6 THEN
		OUT_AG.bRel_IgnOn := OUT_AG.bEng_Start;
	ELSE
		xTON_StartScav(IN:= OUT_AG.bEng_Start, PT:= tiStartScav);
		OUT_AG.bRel_IgnOn := xTON_StartScav.Q;
	END_IF;

	(* set skip fire order for all cylinders while purging *)
	// detect starter demand off after purge cranking cycle
	xF_TRIG_bEleStarter_DemOffPurge(CLK:= bEleStarter_Dem_PurgeCrk);
	IF xEngType.Type6 AND (xF_TRIG_bEleStarter_DemOffPurge.Q AND NOT OUT_AG.tEleStarter_Dem.Do) AND OUT_AG.bMissfCyl_PurgeCrk THEN
		bMissfCyl_AftPurgeCrk := TRUE;
	END_IF;
	IF bMissfCyl_AftPurgeCrk AND IN_AG.rN_EngAct = 0.0 THEN
		bMissfCyl_AftPurgeCrk := FALSE;
	END_IF;

	IF xEngType.Type6 AND ((OUT_AG.bEng_Start AND bEleStarter_Dem_PurgeCrk) OR bMissfCyl_AftPurgeCrk) THEN
		OUT_AG.iMissfCyl_PurgeCrk := xEngType.MisfireOrder[xEngType.NumberOfCylinder];						// switch off all cylinders
		OUT_AG.bMissfCyl_PurgeCrk := TRUE;
	ELSE
		OUT_AG.iMissfCyl_PurgeCrk := 0;
		OUT_AG.bMissfCyl_PurgeCrk := FALSE;
	END_IF;

	(*---------------------------------------------------------------------------------------------*)
	(* Start scavenging monitoring pt.1*)
	xRT_EngRun(CLK:= IN_AG.rN_EngAct > Para.rN_EngStart_LimHiHi);				(* engine running *)

	IF xRT_EngRun.Q AND bStartScavBgn THEN
		bStartScavBgn 			:= FALSE;										(* scavenging at the beginning of the starting procedure trigger reset *)
	END_IF;
	IF xRT_EngRun.Q AND bStartScavBgnFroce THEN
		bStartScavBgnFroce 		:= FALSE;										(* forced anticipated scavenging reset *)
	END_IF;

	IF xRT_EngStart.Q AND (bStartScavFail OR bStartScavBgnFroce) THEN
		bStartScavBgn 			:= TRUE;										(* scavenging at the beginning of the starting procedure activation *)
		bStartScavBgnFroce 		:= FALSE; 										(* forced anticipated scavenging variable reset *)
	END_IF;

	IF (xRT_EngStart.Q AND (M_STRT_TEMP3 OR M_STRT_TEMP4 OR M_STRT_TEMP5) AND NOT bStartScavBgn) THEN 	(* auto or manual starting procedure begins with gas valve open*)
		bStartScavBgnFroce 		:= TRUE; 																(* forced anticipated scavenging set*)
	END_IF;

	(*---------------------------------------------------------------------------------------------*)
	(* start scavenging time with blocked gas valves only during automatic or manual mode *)
	xTON_PostStartScav	(IN:= OUT_AG.bEng_Start, PT:= MAX(xTP_StarterON.PT, xTP_StarterON_Extended.PT + xTON_StarterMeas2.PT + xTP_StarterMeas.PT + bDebugStartActive_Delay) - tiStartScav);	(* GV blocked at the end of starting procedure *)
	xTP_PreStartScav	(IN:= OUT_AG.bEng_Start, PT:= tiStartScav);																																(* GV blocked at the beginning of the starting procedure *)

	IF (NOT xEngType.Type6) AND (M_STRT_TEMP3 OR M_STRT_TEMP4 OR M_STRT_TEMP5) THEN 		(* automatic or manual start procedure *)
		IF	xEngType.Type3 AND NOT bStartScavBgn THEN
			OUT_AG.bGV_Start_ScaveBlock := xTON_PostStartScav.Q;
		ELSIF xEngType.Type3 AND bStartScavBgn THEN
			OUT_AG.bGV_Start_ScaveBlock := xTP_PreStartScav.Q;
		ELSE
			OUT_AG.bGV_Start_ScaveBlock := xTP_PreStartScav.Q AND NOT bCalcAdaptiveStartTime;
		END_IF;
	ELSIF xEngType.Type6 THEN
		OUT_AG.bGV_Start_ScaveBlock := bGV_Block_PurgeCrk;
	ELSE
		OUT_AG.bGV_Start_ScaveBlock := FALSE;
	END_IF;

	(*---------------------------------------------------------------------------------------------*)
	(* Scavenging monitoring pt.2*)
	xR_TRIG_StartScav(CLK := OUT_AG.bEng_Start AND OUT_AG.bGV_Start_ScaveBlock); 	(* beginning of auto or manual start scavenging procedure *)
	xF_TRIG_StartScav(CLK := OUT_AG.bEng_Start AND OUT_AG.bGV_Start_ScaveBlock); 	(* end of auto or manual start scavenging procedure *)

	IF xR_TRIG_StartScav.Q THEN
		bStartScavFail		:= FALSE;												(* scavenging procedure status reset *)
		bStartScavSflMsg	:= FALSE;												(* scavenging procedure failure detection reset *)
		bIgn_Run_CAN_Ok		:= FALSE;												(* ignition system running during scavenging ok reset *)
		bStartScavCmpl		:= FALSE;												(* 10 sec scavenging completed reset *)
	END_IF;

	IF xR_TRIG_StartScav.Q AND bStartScavBgnFroce THEN
		bStartScavBgnFroce := FALSE;												(* forced anticipated scavenging reset *)
	END_IF;

	IF OUT_AG.bEng_Start AND OUT_AG.bGV_Start_ScaveBlock THEN 						(* average speed during auto or manual start scavenging procedure *)
		rN_EngStartScavAvg := (rN_EngStartScavAvg * rCnt_EngStartScavAvg) + IN_AG.rN_EngAct;
		rCnt_EngStartScavAvg := rCnt_EngStartScavAvg + 1;
		IF rCnt_EngStartScavAvg = 95 THEN
			bStartScavCmpl := TRUE;													(* 10 sec scavenging completed *)
		END_IF;
		IF rCnt_EngStartScavAvg > 0 THEN rN_EngStartScavAvg := rN_EngStartScavAvg / rCnt_EngStartScavAvg ; END_IF;
	ELSE
		rCnt_EngStartScavAvg := 0;
	END_IF;

	xTON_Ign_Run_CAN(IN:= OUT_AG.bEng_Start AND OUT_AG.bGV_Start_ScaveBlock AND IN_AG.bIgn_Run_CAN, PT:= T#3s);
	IF OUT_AG.bEng_Start AND OUT_AG.bGV_Start_ScaveBlock THEN
		IF xTON_Ign_Run_CAN.Q THEN
			bIgn_Run_CAN_Ok := TRUE;												(* ignition system running during scavenging for at least 3s *)
		END_IF;
	END_IF;

	IF (xF_TRIG_StartScav.Q AND ((NOT bIgn_Run_CAN_Ok) OR							(* check at the end of auto or manual start scavenging procedure for ignition failure *)
	   (IN_AG.rN_EngAct > Para.rN_EngStart_LimHi) OR								(* or engine starting during scavenging *)
	   (rN_EngStartScavAvg < Para.rN_EngStartMon_LimHi) OR							(* or insufficient average speed reached at the end of scavenging *)
		NOT bStartScavCmpl)) THEN													(* or 10 sec scavenging not completed *)
		bStartScavFail := TRUE;														(* scavenging procedure failure *)
	END_IF;

	IF xEngType.Type3 AND xF_TRIG_StartScav.Q AND NOT bStartScavFail THEN			(* scavenging by starting system successful B9088 *)
		bStartScavSflMsg 	:= TRUE;
	END_IF;

	IF xEngType.Type3 AND bStartScavBgn AND bStartScavFail THEN						(* unsuccessful scavenging by starting system A2376 *)
		bStartScavUnsfl		:= TRUE;
	END_IF;

	(*---------------------------------------------------------------------------------------------*)
	(* start time  statistics *)
	usStatus_gettime	:= RTC_gettime(ADR(tGetTime));			(* FuB aktuelle Zeit einlesen *)

	IF xRT_EngStart.Q THEN
		tiStartTime := tGetTime;
	END_IF;

	IF xF_TRIG_StarterMeas.Q THEN								(* Start speed measurement done *)
		Perm.tStartStat[Perm.StatCnt].tiStarterON_Max :=	ti_EngStart_Max;
		Perm.tStartStat[Perm.StatCnt].tiStartScav :=		tiStartScav;
		Perm.tStartStat[Perm.StatCnt].rN_EngStart :=		rN_EngStart;
	END_IF;

	IF xFT_EngStart.Q THEN
		Perm.tStartStat[Perm.StatCnt].tiStartTime := 		tGetTime;

		Perm.tStartStat[Perm.StatCnt].tiStartDuration := UDINT_TO_TIME((USINT_TO_UDINT(tGetTime.hour)*3600000 + tGetTime.minute * 60000 + tGetTime.second * 1000 + tGetTime.millisec)
		- (tiStartTime.hour*3600000 + tiStartTime.minute*60000 + tiStartTime.second*1000 + tiStartTime.millisec));	(* actual used time to start *)
		MM2VIS.rTi_EngStart_Duration := TIME_TO_REAL(Perm.tStartStat[Perm.StatCnt].tiStartDuration) ;

		IF IN_AG.iCnt_Starts > 0 THEN
			Perm.tStartStat[Perm.StatCnt].iStartID :=		IN_AG.iCnt_Starts;									(* BENÖTIGT ZUSÄTZLICHES MODULINTERFACE! *)
		ELSE
			Perm.tStartStat[Perm.StatCnt].iStartID := 		(Perm.StatCnt + REAL_TO_DINT(Perm.rAG_PermValue1));	(*=Backuplösung bei fehlender Modulinterfaceerweiterung: in PermValue1 einmalig den korr. Startzählerstand eingeben *)
		END_IF;
		Perm.tStartStat[Perm.StatCnt].bStartSuccess :=		(IN_AG.rN_EngAct > (rN_EngStart * 1.1));	(* simplified condition to detect start ok -> TO VERIFY on pilot engines! *)
		Perm.tStartStat[Perm.StatCnt].tiStarterOFF :=		tiStarterOFF;
		Perm.StatCnt := 	Perm.StatCnt +1;
		IF Perm.StatCnt > 200 THEN Perm.StatCnt := 0; END_IF;

		MM2VIS.rTi_EngStart_Delay := TIME_TO_REAL(tiStarterOFF);
	END_IF;

	(*---------------------------------------------------------------------------------------------*)
	(* demand mains start device *)
	OUT_AG.tMainsStartDevDem.Do := IN_AG.bEng_Dem AND NOT IN_AG.tEng_Run.Do;

END_PROGRAM
```

#### EleStart.var
```iecst
VAR
	M_STRT_TEMP3 : BOOL;
	M_STRT_TEMP4 : BOOL;
	M_STRT_TEMP5 : BOOL;
	M_STRT_TEMP6 : BOOL;
	M_STRT_TEMP7 : BOOL;
	T7_TEMP1 : BOOL;
	xCTD_Start : CTD;
	xR_TRIG_AutoStartErr : R_TRIG;
	xR_TRIG_Reset1 : R_TRIG;
	xR_TRIG_Reset2 : R_TRIG;
	xR_TRIG_Reset3 : R_TRIG;
	xR_TRIG_Reset4 : R_TRIG;
	xF_TRIG_Start : F_TRIG;
	xTOF_LockAckStarter : TOF;
	xTON_StartErr : TON;
	xTON_StartScav : TON;
	xTON_ChargeOff : TON;
	xTON_H_STRT : TON;
	xTON_DelayStart : TON;
	xTON_Reset4 : TON;
	xTON_ZAZ : TON;
	xTP_StarterON : TP;
	xTP_StarterOFF : TP;
	ZM_HSTART : BOOL;
	xTON_DelayManStart : TON;
	xTP_StarterMeas : TP;
	bCalcAdaptiveStartTime : BOOL;
	rN_EngStartAvg : REAL;
	rCnt_EngStartAvg : REAL; (*internal use only: avarage counter*)
	xF_TRIG_StarterMeas : F_TRIG;
	rTiFactor_Cylinders : REAL;
	rTiFactor_N_EngStart : REAL;
	LCRScal_Cylinders : LCRScal;
	LCRScal_N_EngStart : LCRScal;
	tiStarterON1 : TIME; (*Testbench ONLY*)
	tiStarterON2 : TIME; (*Testbench ONLY*)
	tiStarterON3 : TIME; (*Testbench ONLY*)
	tiStarterOFF1 : TIME; (*Testbench ONLY*)
	tiStarterOFF2 : TIME; (*Testbench ONLY*)
	tiStarterOFF3 : TIME; (*Testbench ONLY*)
	tiStartScav1 : TIME; (*Testbench ONLY*)
	tiStartScav2 : TIME; (*Testbench ONLY*)
	tiStartScav3 : TIME; (*Testbench ONLY*)
	tiStarterON_Base : TIME;
	bDebugStartActive : BOOL;
	tiStartScav : TIME;
	tiStarterOFF : TIME;
	xTON_StarterMeas2 : TON;
	xTP_PreStartScav : TP; (*scavenging at the beginning of the start attempt*)
	xTON_PostStartScav : TON; (*scavenging at the end of the start attempt*)
	bDebugTON_StarterMeas2 : BOOL;
	bTriggerStarterMeas : BOOL;
	tiStarterON_Max : TIME;
	xTP_StarterON_Extended : TP;
	bTP_StarterON : BOOL;
	ti_EngStart_Max : TIME;
	usStatus_gettime : UINT;
	tGetTime : RTCtime_typ;
	tiStartTime : RTCtime_typ;
	xRT_EngStart : R_TRIG;
	xFT_EngStart : F_TRIG;
	xRT_EngRun : R_TRIG; (*Engine running*)
	rN_EngStart : REAL; (*Display Value of start speed*)
	rN_EngStartScavAvg : REAL; (*Average engine speed during scavenging*)
	rCnt_EngStartScavAvg : REAL; (*internal use only: avarage speed scavenging counter*)
	bAdoptiveStartEnab : BOOL; (*Activation bit for whole new start process*)
	rStarterON_Max : REAL; (*internal*)
	xR_TRIG_StartScav : R_TRIG; (*beginning of scavenging*)
	xF_TRIG_StartScav : F_TRIG; (*end of scavenging*)
	xRT_bDebugStartActive : R_TRIG; (*extended starting time calculation enabled*)
	bDebugStartActive_Delay : TIME; (*detect turning starter delay*)
	xTON_Ign_Run_CAN : TON; (*ignition system running during scavenging for 3s*)
	bIgn_Run_CAN_Ok : BOOL; (*ignition system running during scavenging ok*)
	bStartScavCmpl : BOOL; (*10 sec scavenging completed*)
	xTON_EleStarter_Mon : TON; (*starter/s correct engagement monitoring trigger*)
	xTP_EleStarter_Mon : TP; (*timer for voltage measurement*)
	xFT_EleStarter_Mon : F_TRIG; (*correct engagement monitoring evaluation instant*)
	rU_EleStarterAvg1 : REAL; (*starter 1 terminal 45 average voltage*)
	rU_EleStarterAvg2 : REAL; (*starter 2 terminal 45 average voltage*)
	rU_EleStarterAvg3 : REAL; (*starter 3 terminal 45 average voltage*)
	rCnt_EleStarterAvg : REAL; (*internal use only: starter terminal 45 average voltage counter*)
	b_EleStarter_EngageFail : BOOL; (*starters did not engage*)
	iVolFlow_RunEng : UDINT; (*volume flow through the engine [lt/s]*)
	rVol_CylDis : REAL; (*Single cylinder displacement [lt]*)
	rVolFlow_RunEng : REAL; (*volume flow through the engine [lt/s]*)
	rVol_PurgeAir : REAL; (*Volume of purge air [lt]*)
	xTON_GVOpen_1s : TON; (*Gas valve open for more than 1 second*)
	tiCycleTime : TIME; (*task cycle time*)
	rCycleTime : REAL; (*task cycle time, real variable in seconds*)
	RTInfo_CTR : RTInfo;
	xF_TRIG_bEleStarter_Dem : F_TRIG; (*detect beginning of starter cool down phase*)
	rTi_ST_Active : REAL; (*cumulated starting time [s]*)
	rTi_ST_Active_zero : REAL; (*cumulated starting time at the beginning of cool down phase [s]*)
	rTi_ST_Cooldown : REAL; (*starter cood down phase duration [s]*)
	rTi_ST_Res : REAL; (*remaining starting time[s]*)
	xGR_MINR_bSt_STT : GR_MINR; (*starter temperature status*)
	bSt_STT : BOOL; (*starter temperature status (TRUE: not overheated, FALSE: overheated)*)
	bReq_Rel_STT : BOOL; (*request for the starter temperature release*)
	bReq_Rel_STT_PurgeCrk : BOOL; (*request from the purge cranking cycle for the starter temperature release*)
	bRel_STT_Ena : BOOL; (*Starter temperature release function enabled*)
	bSt_RelAuxOff_STT : BOOL; (*starter temperature release off*)
	rTi_ST_Active_AftCooldown : REAL; (*cumulated starting time after cooldown phase [s]*)
	rTi_ST_UntRelDur : REAL; (*time duration until starter temperature release [s]*)
	bReq_PurgeCrk : BOOL; (*purge cranking cycle request*)
	bPurgeCrk_Run : BOOL; (*purge cranking cycle running*)
	bGV_Block_PurgeCrk : BOOL; (*purge cranking cycle GV blocked*)
	xR_TRIG_bSt_Purge : R_TRIG; (*purge cranking cycle successful rising egde*)
	bDem_ST_PurgeCrk : BOOL; (*demand starter from purge cranking cycle *)
	bEleStarter_Dem_PurgeCrk : BOOL; (*starter demanded and released from purge cranking cycle *)
	rFuelAdm : REAL; (*fuel admission status*)
	rVol_Mx : REAL; (*volume of mixture [lt]*)
	xR_TRIG_bReq_StartAtt : R_TRIG; (*request for start attempt rising edge*)
	bReq_StartAtt : BOOL; (*request for start attempt*)
	bRel_STT_StartAtt : BOOL; (*release from starter temperature for start attempt*)
	bStartAtt_Run : BOOL; (*start attempt running*)
	bDem_ST_StartAtt : BOOL; (*demand starter from start attempt*)
	rTiStartAttDur : REAL; (*start attempt duration*)
	xR_TRIG_bReq_Rel_STT_StartAtt : R_TRIG; (*request release from starter temperature for start attempt*)
	xTON_bSt_RelAuxOff_STT : TON; (*starter temperature release off delay before setting message*)
	xGR_MAXR_SpeedMon : GR_MAXR; (*detect filtered speed drop below 50 rpm*)
	xF_TRIG_SpeedMon : F_TRIG; (*detect filtered speed drop below 50 rpm*)
	bSpeedMon_PurgeCrkStartAtt : BOOL; (*Speed monioring status during purge cranking cycle and start attempt (true: unsuccessfull, false, successful)*)
	bEng_SU_Man_Req : BOOL; (*Manual startup released and requested *)
	bEleStarter_Dem_StartAtt : BOOL; (*starter demanded and released from start attempt*)
	bRel_Nospeed : BOOL; (*starter released when no speed*)
	xF_TRIG_bEng_Dem_EPS : F_TRIG; (*emergency operation demand reset*)
	bFS_Req : BOOL; (*Fast start requested*)
	xR_TRIG_bParaSetupOk : R_TRIG; (*parameter set up rising edge*)
	xF_TRIG_bSt_RelAuxOff_STT : F_TRIG; (*starter temperature release off falling edge*)
	xF_TRIG_GVopen_bEGScavAct : F_TRIG; (*Gas valve open and EG scavenging active falling edge*)
	xF_TRIG_bEleStarter_DemOffPurge : F_TRIG; (*EleStarter demand after purge cranking cylce falling edge*)
	bMissfCyl_AftPurgeCrk : BOOL; (*Skip fire order after purge cranking cycle*)
	xTP_bSfl_PurgeCrk : TP; (*Purge cranking cycle successfull TP*)
	iVol_MinAirLim_SysPurge : UDINT; (*Limited minimum air volume required for system purge *)
	xTON_Nospeed15s : TON; (*zero speed for 15 s*)
END_VAR
```

### Program Logical/AuxiliariesGeneral/AirStart (IEC, version 4.10.0) - air start

#### AirStartCyclic.st - Cyclic code
```iecst
(****************************************************************************************************************************************
AirStart		pressurized air starters (CYCLIC)

This code is confidential AND proprietary to the INNIO Company.
It may NOT be used in any form, or reproduced in any manner,
without the express written permission of the INNIO Company.
Copyright, INNIO Company, 2019

Customized modifications: -
------------------------

History:
-------
V3.20.0	26.07.2010 koppm.	new
		13.08.2010 koppm.	slowturn wieder freigegeben
		25.10.2012 TinelloM	Nach einem SlowTurn muss die Drehzahl zuerst wieder unter 14 Umdrehungen gehen, bevor durchgestartet wird.
							Pausenzeit zwischen Slowturn und Durchstarten der Maschine im INIT
V3.50.0	22.10.2013 TinelloM	added  NOT xTON_SlowturnPassed.Q
							added bRelEngTurn_OilSkid
		08.04.2014 lettenb.	xTON_O2Start_M: FGDRPS added
V3.59.0 30.12.2014 TinelloM	New Spezi; Anpassung an XT4
V4.00.0	06.02.2015 Walid Mari Code-Portierung in XT4
V4.00.1 18.03.2015 lettenb.	bugfix (sky global ib) / Release monitoring -> NOT entfernt
		21.05.2015 lettenb.	rCnt_N_AirStarterOld > iCnt_N_AirStarterOld (REAL > DINT) TO avoid overflow(tinello)
							OUT_AG.bSlowturn_Active added FOR statistics
V4.03.0 17.09.2015 			M_STRT_TEMP6/7: starter ON FOR N2 scavenging + ignition selftest added
V4.04.0	29.06.2016 TinelloM	trip prevention in CASE OF starter stop
		18.11.2016 TinelloM	xTON_DelayStart.PT, xTON_DelayManStart.PT: 6->0s start delay removed(fahringer)
		18.01.2017 TinelloM airstarter speed convert TO UINT
V4.05.0 21.04.2017 lettenb.	airstarter SWAT920/2.2
V4.05.1 14.06.2017 lettenb.	fast start added
V4.05.1 14.12.2017 lettenb.	spare para removed
V4.07.0 26.04.2018 lettenb.	slowturn removed, SWAT920/5
        13.06.2018 lettenb.	IN_AG.bFS_Act := TRUE -> FALSE; // activation only for 30s faststart, with 4 starters and preengagement
		29.06.2018			bFS4_Act added, 4 starters configuration
V4.09.0	11.12.2019 Schmid	new air starter logic
V4.10.0	29.01.2021 Schmid	manual start stop buttons from Opstate instead of VIS

Instructions FOR use:
--------------------

Outstandings:
------------
bFS4_Act parameter ? standardization 4 starters variant ?
renaming Do's for 4 starter configuration
(****************************************************************************************************************************************)
PROGRAM _CYCLIC

	IF NOT xEngType.Type9 THEN RETURN;		(* Avoid running Airstart and EleStart in same time *)
	END_IF;

	(*--------------------------------------------------------------*)
	(* RESET of alarms and warnings 								*)
	(*--------------------------------------------------------------*)
	bAMM_Pr_AirStarter_Tank_Ms		:= FALSE;
	bAMM_Pr_AirStarter_Tank_Lo		:= FALSE;
	bAMM_Pr_AirStarter_Tank_LoLo	:= FALSE;

	bAMM_Pr_AirStarter_Supply_MsMs	:= FALSE;
	bAMM_Pr_AirStarter_Supply_LoLo	:= FALSE;
	bAMM_Pr_AirStarter_Supply_HiHi	:= FALSE;

	bAMM_AirStarter_StartUp			:= FALSE;

	bAMM_Pr_AirST_Engage_Lo			:= FALSE;
	bAMM_Pr_AirST_Engage_Ms			:= FALSE;

	(* air starter speed [rpm]							E.00-SI-006 *)
	IF xEngType.NumberOfTeeth > 0 THEN (* 920: 398 *)

		iN_AirSt  	  	:= DINT_TO_UINT(IN_AG.tCnt_N_AirStarter.Ai);

		IF iN_AirSt >= iN_AirSt_old THEN	iN_AirStDiff	:= iN_AirSt - iN_AirSt_old;
									ELSE	iN_AirStDiff	:= (65535   - iN_AirSt_old) + iN_AirSt;
		END_IF;

		rN_AirStarter 	:= LIMIT(0, UINT_TO_REAL(iN_AirStDiff) * 300 / UINT_TO_REAL(xEngType.NumberOfTeeth), 2000);
												(* 300 = 600(Umrechnung von 100ms auf min) : 2(jede Flanke wird gezählt)	*)
 	ELSE
 		rN_AirStarter 	:= 0;
 	END_IF;

	iN_AirSt_old 		:= DINT_TO_UINT(IN_AG.tCnt_N_AirStarter.Ai);

	(* check fly wheel movement with: *)
	IF OUT_AG.tAirST_ValEngage.Do THEN
		(* count gear slopes (teeth) that the starter speed sensor detects during engagement phase *)
		iCnt_AirST_MovingFlyW := iCnt_AirST_MovingFlyW + iN_AirStDiff;

		(* if number does not change for >1min: trigger reset of tooth counter *)
		IF iCnt_AirST_MovingFlyW <> iCnt_AirST_MovingFlyW_old THEN
			iCnt_AirST_MovingFlyW_old	 := iCnt_AirST_MovingFlyW;
			xTON_MovingFlyW_Cnt_Reset.IN := FALSE;
		ELSE
			xTON_MovingFlyW_Cnt_Reset.IN := NOT xTON_MovingFlyW_Cnt_Reset.Q;
		END_IF;

		(* reset tooth counter *)
		IF xTON_MovingFlyW_Cnt_Reset.Q THEN
			iCnt_AirST_MovingFlyW		:= 0;
			iCnt_AirST_MovingFlyW_old	:= 0;
		END_IF;

	(* reset tooth counter after engine start or no engagement command *)
	ELSIF NOT bComEngage THEN
		iCnt_AirST_MovingFlyW		 := 0;
		iCnt_AirST_MovingFlyW_old	 := 0;
		xTON_MovingFlyW_Cnt_Reset.IN := FALSE;
	END_IF;

	xTON_MovingFlyW_Cnt_Reset.PT	:= T#1m;
	xTON_MovingFlyW_Cnt_Reset();

	bAirST_Engaged_MovingFlyW	:= (iCnt_AirST_MovingFlyW > 8);		(* tolerate movement of up to 4 teeth (8 gear slopes) during engagement *)

	(* end check fly wheel movement *)

	(****************************************************************************************************************************************************)
	(************************         		     					  error monitoring		 	       		      	           **************************)
	(****************************************************************************************************************************************************)
	IF IN_AG.tPB2MM.bParaSetupOk THEN

		(* measurement signal failure 								*)
		bAMM_Pr_AirStarter_Tank_Ms			:= Para.bPr_AirStarter_Tank_Exist 	AND NOT IN_AG.tPr_AirStarter_Tank.GoodQual;						(* W2559 *)
		bAMM_Pr_AirStarter_Supply_MsMs		:= Para.bPr_AirStarter_Supply_Exist	AND NOT IN_AG.tPr_AirStarter_Supply.GoodQual AND NOT M_DREHZ;	(* W2557 - was A3370 -> desensitized *)
		xTON_Pr_AirST_Engage_Ms(IN:= NOT IN_AG.tPr_AirST_Engage.GoodQual, PT:= T#1s);
		bAMM_Pr_AirST_Engage_Ms				:= xTON_Pr_AirST_Engage_Ms.Q;																		(* W9303 *)

		(* release monitoring	*)
		xTOF_Pr_AirStarter_Tank(IN	:= bAMM_Pr_AirStarter_Tank_Ms, 		PT:= T#10s);		(* TOF because of filtered signals *)
		xTOF_Pr_AirStarter_Supply(IN:= bAMM_Pr_AirStarter_Supply_MsMs, 	PT:= T#10s);

		bRelMon_Pr_AirStarter_Tank		:= Para.bPr_AirStarter_Tank_Exist	AND NOT xTOF_Pr_AirStarter_Tank.Q;
		bRelMon_Pr_AirStarter_Supply	:= Para.bPr_AirStarter_Supply_Exist	AND NOT xTOF_Pr_AirStarter_Supply.Q;

		(* tank pressure											*)
		IF M_DREHZ THEN bAMM_Pr_AirStarter_Tank_Lo	 := (IN_AG.tPr_AirStarter_Tank.Ai < Para.rPr_AirStarter_Tank_Lo) AND bRelMon_Pr_AirStarter_Tank;		(* W2560 *)
		ELSE			bAMM_Pr_AirStarter_Tank_LoLo := (IN_AG.tPr_AirStarter_Tank.Ai < Para.rPr_AirStarter_Tank_Lo) AND bRelMon_Pr_AirStarter_Tank;		(* A2268 *)
		END_IF;

		(* supply pressure											*)
		IF NOT M_DREHZ AND bRelMon_Pr_AirStarter_Supply THEN
			bAMM_Pr_AirStarter_Supply_LoLo	:= (IN_AG.tPr_AirStarter_Supply.Ai < Para.rPr_AirStarter_Supply_LoLo);								(* A2269 *)
			bAMM_Pr_AirStarter_Supply_HiHi	:= (IN_AG.tPr_AirStarter_Supply.Ai > Para.rPr_AirStarter_Supply_HiHi);								(* A2267 *)
		END_IF;

		(* engagement pressure sensor											*)
		bPr_AirST_Engage_Lo := (IN_AG.tPr_AirST_Engage.Ai < 5.0);
		xTON_Pr_AirST_Engage_Lo(IN:= OUT_AG.tAirST_ValEngage.Do AND bPr_AirST_Engage_Lo, PT:= T#2s);
		bAMM_Pr_AirST_Engage_Lo		:= xTON_Pr_AirST_Engage_Lo.Q;			(* W2425 air starter engaging error - pressure at pressure sensor low*)

		IF Para.bN_AirStarter_Exist THEN
			(* starter engagement condition dep. on OMSS ----------*)
			IF		bOMSS_Aut THEN	bAirST_Engage_OMSS :=	TRUE;				(* pre-engagement for fast start *)
			ELSIF	bOMSS_Man THEN	bAirST_Engage_OMSS :=	IN_AG.bEng_Aux_Dem;	(* engagement with start preparation *)
			ELSIF	bOMSS_Off THEN	bAirST_Engage_OMSS :=	M_STRT_TEMP7;		(* start scavenging request from ignition selftest *)
			ELSE  					bAirST_Engage_OMSS :=	FALSE;
			END_IF;

			(* starter engagement command -------------------------*)
			bComEngage :=	bAirST_Engage_OMSS
						AND NOT M_DREHZ
						AND NOT bGnlTrip
						AND NOT IN_AG.bEng_Bloc;

			IF EDGEPOS(bComEngage) THEN
				iStepCnt 		:= 10;
				iCntEng			:= 0;
			ELSIF NOT bComEngage THEN
				iStepCnt 		:= 0;
				iCntEng			:= 0;
			END_IF;

			xTON_EngStop(IN:= ((IN_AG.rN_EngAct < 0.1) AND (rN_AirStarter < 0.1)), PT:= T#10s); //engine stopped

		(*----------------------------------------------------------------*)
			CASE iStepCnt OF
				0:	bAirST_ValEngage	:= FALSE;
					bAirST_ValStart	:= FALSE;
					bAMM_EngageErr			:= FALSE;
					xTON_AirST_ValEngage(IN:= FALSE, PT:= T#0s);
					xTON_AirST_ValEngageOff(IN:= FALSE, PT:= T#0s);

				10: (* Step 1: Open engagement valve *)
					xTON_AirST_ValEngage(IN:= bAirST_ValEngage, PT:= T#2s);
					bAirST_ValEngage := xTON_EngStop.Q OR bAirST_ValEngage;
					IF xTON_AirST_ValEngage.Q THEN
						iStepCnt := iStepCnt + 10;
						xTON_AirST_ValEngage(IN:= FALSE, PT:= T#0s);//reset ton
					END_IF;

				20: (* Step 2: Check engagement pressure *)
					IF NOT bPr_AirST_Engage_Lo AND bAirST_ValEngage THEN
							iStepCnt := iStepCnt + 10;
					ELSE
						xTON_AirST_ValEngageOff(IN:= NOT bAirST_ValEngage, PT:= Para.tiReEngage);
						bAirST_ValEngage := FALSE;
						IF xTON_AirST_ValEngageOff.Q THEN
								iStepCnt := iStepCnt + 1; //repeat_engagement ?;
								iCntEng  := iCntEng  + 1;
								xTON_AirST_ValEngageOff(IN:= FALSE, PT:= T#0s); //reset ton
						END_IF;
					END_IF;

				21: (* Step 2.1: Further engagement attempt *)
					IF (iCntEng >= 3)			THEN bAMM_EngageErr := TRUE;  END_IF;	//A3375
					IF (rN_AirStarter > 0.0)	THEN bAMM_EngageErr := TRUE;  END_IF;	//A3375
					IF (IN_AG.rN_EngAct > 0.0)	THEN bAMM_EngageErr := TRUE; 	        //A3375
					ELSE iStepCnt := 10;											//next engagement
					END_IF;

				30: (* Step 3: Move check/waiting for start command *)
					IF (bAirST_Engaged_MovingFlyW OR (IN_AG.rN_EngAct > 0.0))	THEN bAMM_EngageErr := TRUE;			//A3375
					ELSIF bPr_AirST_Engage_Lo									THEN bAMM_Pr_AirST_Engage_Lo := TRUE;	//W2425
																					 iStepCnt := 20;
					ELSIF OUT_AG.bEng_Start										THEN bAirST_ValStart := TRUE;
																					 iStepCnt := iStepCnt + 10;
					END_IF;

				40: (* Step 4: Check starter speed up *)
					IF (IN_AG.tEng_Run.Do OR M_DREHZ) THEN iStepCnt := 0;
					ELSE
						bAirST_ValStart := OUT_AG.bEng_Start AND NOT xTP_AirST_ValStart_Interrupt.Q;
					END_IF;

				ELSE iStepCnt := 0;
			END_CASE;

		END_IF;

		(*----------------------------------------------------------*)
		(* start up failure	*)
		xTON_FailedAirST(IN:= (rN_AirStarter < 40) AND OUT_AG.tAirST_ValStart.Do AND OUT_AG.bEng_Start, PT:= Para.tiAirST_Interrupt);
		xTP_AirST_ValStart_Interrupt(IN:= xTON_FailedAirST.Q AND (IN_AG.rN_EngAct < 40.0), PT:= T#1s);

		(* safi safety loop *)
		xTOF_STP_STRT(IN:= OUT_AG.bEng_Start AND (xTON_FailedAirST.Q OR xTOF_STP_STRT.IN), PT:= T#10s);
		OUT_AG.STP_STRT := xTOF_STP_STRT.Q;

		xF_TRIG_Eng_Start(CLK:= OUT_AG.bEng_Start);
		IF EDGEPOS(xTP_AirST_ValStart_Interrupt.Q)	THEN iCntSt := iCntSt + 1; (* 3 start up (N > 40 rpm) attempts *)
		ELSIF (RESET OR xF_TRIG_Eng_Start.Q)		THEN iCntSt := 0;
		END_IF;

		bAMM_AirStarter_StartUp   := OUT_AG.bEng_Start AND (IN_AG.rN_EngAct < 40) AND (iCntSt >= 3); (* A3369 startup failure air starter            (N<40)*)

	END_IF;

	(****************************************************************************************************************************************************)
	(************************         		     			Handling of starter - similar to EleStart  				           **************************)
	(****************************************************************************************************************************************************)
	(* start stop button info from Opstate *)
	bStart 	:= IN_AG.bStart;
	bStop 	:= IN_AG.bStop;

	(* delay automatic start *)
	xTON_DelayStart(IN:= IN_AG.bEng_SU_Aut AND NOT bOMSS_Man, PT:= T#0s);
	OUT_AG.bEngAutStartDelay := xTON_DelayStart.Q;

	(* second button push in manual start after short 120s prelubrication time *)
	IF bStart AND xTOF_ShortPreLubeTime_Delay.Q 	THEN ZM_bStartMan := TRUE;
	ELSIF ZM_HSTART	OR NOT IN_AG.bEng_Dem			THEN ZM_bStartMan := FALSE;
	END_IF;

	(* manual start *)
	ZM_HSTART	:= 	(bStart OR ZM_HSTART OR ZM_bStartMan)
			AND		bOMSS_Man
			AND 	(AN_VSD1 OR AN_VSD2)
			AND 	bPr_OTC_Prelub
			AND 	IN_AG.bEng_SU_Man
			AND(NOT IN_AG.bBlocDelay_ManStart OR     OUT_AG.bEng_Start)
			AND    	(IN_AG.bScavFinished      OR NOT IN_AG.bRel_ScavN2)
			AND NOT xTP_StarterOFF.Q
			AND NOT bStop;

	(* delay manual start *)
	xTON_DelayManStart(IN:= ZM_HSTART AND bOMSS_Man, PT:= T#0s);

	(* starter pulse ON-time *)
	T7_TEMP1 := (IN_AG.bEng_Dem_EPS AND NOT IN_AG.bOnly_Island) OR OUT_AG.bEngAutStartDelay;
	xTP_StarterON.PT := Para.tiAirStarter_OnTime;

	IF NOT IN_AG.bEng_Dem_EPS AND NOT ZM_HSTART AND NOT IN_AG.bEng_SU_Aut THEN (* reset timer *)
		xTP_StarterON(IN:= FALSE, PT:= T#0s);
	ELSIF IN_AG.bEng_SU_Man THEN
		xTP_StarterON(IN:= xTON_DelayManStart.Q AND NOT xTP_StarterOFF.Q);
	ELSIF IN_AG.bEng_SU_Aut THEN
		xTP_StarterON(IN:= T7_TEMP1             AND NOT xTP_StarterOFF.Q);
	ELSE
		xTP_StarterON(IN:= FALSE, PT:= T#0s);
	END_IF;
	bTP_StarterON := xTP_StarterON.Q ;

	(* starter puls OFF-time *)
	xTP_StarterOFF(IN:= NOT bTP_StarterON, PT:= T#60s);

	(*---------------------------------------------------------------------------------------------*)
	(* monitoring start *)
	xR_TRIG_Reset1(CLK:= IN_AG.tEng_Run.Do);
	xR_TRIG_Reset2(CLK:= IN_AG.bEng_Dem_Man_SUpF);
	xR_TRIG_Reset3(CLK:= IN_AG.bEng_Dem_Aut_SUpF);
	RESET := xR_TRIG_Reset1.Q OR xR_TRIG_Reset2.Q OR xR_TRIG_Reset3.Q;

	xF_TRIG_Start(CLK:= bTP_StarterON);

	(* start counter *)
	xCTD_Start(CD:= xF_TRIG_Start.Q, LOAD:= RESET, PV:= 3);
	OUT_AG.iStartCount	:= LIMIT(1, xCTD_Start.PV - xCTD_Start.CV + 1, xCTD_Start.PV);  //Number of Start for OpState

	(* man + auto start error *)
	xTON_StartErr(IN:= xCTD_Start.Q AND NOT M_DREHZ AND(IN_AG.bEng_Dem_Aut_SUpF OR IN_AG.bEng_Dem_Man_SUpF), PT:= T#12s); (* delay = min.starter off interval time *)
	bStartErr := xTON_StartErr.Q AND NOT MM2VIS.bMsg3369;		(* A1023 engine start up failure (n>40)*)

	(*---------------------------------------------------------------------------------------------*)
	(* starter ON for N2 scavenging *) (* -> NOT ACTIVE FOR NOW *)
	M_STRT_TEMP6 := IN_AG.bN2_ScavCoStarterOn  AND IN_AG.bRel_ScavN2
				AND OUT_AG.bPr_EOP_Prelub1 AND IN_AG.bRelEngTurn_OilSkid AND NOT M_DREHZ;

	(* starter ON for ignition selftest *)
	M_STRT_TEMP7 := IN_AG.b_ST_DemIgn
				AND OUT_AG.bPr_EOP_Prelub1 AND IN_AG.bRelEngTurn_OilSkid AND NOT M_DREHZ;

	(*---------------------------------------------------------------------------------------------*)
	(* start *)
	ZM_STRT   := IN_AG.bEng_Rel AND NOT M_DREHZ AND OUT_AG.bRelEngOp_Aux;
	OUT_AG.bEng_Start := (ZM_STRT AND bTP_StarterON) 						(* Equal to M_STRT in XT3 *)
//					  OR  M_STRT_TEMP6
					  OR  M_STRT_TEMP7;

	(*---------------------------------------------------------------------------------------------*)
	(* start scavenging time with blocked ignition -> no scavenging for 920 *)
	OUT_AG.bRel_IgnOn := OUT_AG.bEng_Start;

	(* start scavenging time with blocked gas valves -> no scavenging for 920 *)
	OUT_AG.bGV_Start_ScaveBlock := FALSE;

	(* disable direct air injection on starter tank pressure low*)
	OUT_AG.bAMM_Pr_AirStarter_Tank_Lo := bAMM_Pr_AirStarter_Tank_Lo;

	(* safi safety loop - thooth to thooth/engagement failed *)
//	xTOF_STP_STRT(IN:= OUT_AG.bEng_Start, PT:= T#15s);
//	OUT_AG.STP_STRT	:= xTOF_STP_STRT.Q;
//	xTON_ZAZ(IN := OUT_AG.tAirStarter_ValveOn.Do AND (IN_AG.rN_EngAct < 40), PT:= Para.tiReEngage);
//	OUT_AG.STP_STRT := xTON_ZAZ.Q OR ;

	(****************************************************************************************************************************************************)
	(************************              						 air starter valves		 	             			           **************************)
	(****************************************************************************************************************************************************)
	OUT_AG.tAirST_ValEngage.Do	:=  bAirST_ValEngage; 					(* engaging valve    *)
	OUT_AG.tAirST_ValStart.Do	:=  bAirST_ValStart; 	 				(* start    valve    *)

	(****************************************************************************************************************************************************)
	(************************      		        	RELEASE of engine turn equipment (Durchdrehvorrichtung)   			       **************************)
	(****************************************************************************************************************************************************)
	xTON_TURN(IN:= NOT IN_AG.bEng_RPSDem AND NOT IN_AG.bGV_On, PT:= T#1m);  	(* No release of barring gear if engine demand or gasvalve opened *)
	OUT_AG.tTurnRel.Do	:= xTON_TURN.Q AND IN_AG.bRelEngTurn_OilSkid;

END_PROGRAM
```

#### AirStart.var - Local variables
```iecst
VAR
	bRelMon_Pr_AirStarter_Supply : BOOL := FALSE; (*Release monitoring air starter tank pressure *)
	bRelMon_Pr_AirStarter_Tank : BOOL := FALSE; (*Release monitoring air starter supply pressure *)
	bTP_StarterON : BOOL;
	iN_AirSt : UINT; (*Actual value from air starter speed counter*)
	iN_AirStDiff : UINT; (*Difference (Actual - Last) value from air starter speed counter*)
	iN_AirSt_old : UINT; (*Last value from air starter speed counter*)
	M_STRT_TEMP6 : BOOL;
	M_STRT_TEMP7 : BOOL;
	T7_TEMP1 : BOOL;
	xCTD_Start : CTD;
	xF_TRIG_Start : F_TRIG;
	xR_TRIG_Reset1 : R_TRIG;
	xR_TRIG_Reset2 : R_TRIG;
	xR_TRIG_Reset3 : R_TRIG;
	xTOF_Pr_AirStarter_Supply : TOF := (0);
	xTOF_Pr_AirStarter_Tank : TOF := (0);
	xTON_DelayManStart : TON;
	xTON_DelayStart : TON;
	xTON_Pr_AirST_Engage_Lo : TON := (0);
	xTON_StartErr : TON;
	xTON_TURN : TON;
	xTP_StarterOFF : TP;
	xTP_StarterON : TP;
	xTOF_STP_STRT : TOF;
	ZM_HSTART : BOOL;
	xTON_FailedAirST : TON;
	iCntSt : UINT;
	bAirST_Engaged_MovingFlyW : BOOL;
	iCnt_AirST_MovingFlyW : INT := (0);
	iCnt_AirST_MovingFlyW_old : INT := (0);
	xTON_MovingFlyW_Cnt_Reset : TON;
	bComEngage : BOOL;
	bAirST_Engage_OMSS : BOOL;
	iStepCnt : INT := (0);
	iCntEng : INT := (0);
	xTON_AirST_ValEngage : TON;
	xTON_AirST_ValEngageOff : TON;
	xTON_EngStop : TON := (0);
	ZM_bStartMan : BOOL; (* ZM - Start Manual *)
	bPr_AirST_Engage_Lo : BOOL;
	xTP_AirST_ValStart_Interrupt : TP;
	xF_TRIG_Eng_Start : F_TRIG;
	xTON_Pr_AirST_Engage_Ms : TON;
	bAirST_ValEngage : BOOL; (*Command air starter engagement valve (E.31-YCS-001)*)
	bAirST_ValStart : BOOL; (*Command air starter start valve (E.31-YCS-002)*)
END_VAR
```

### Program Logical/AuxiliariesGeneral/blowby (IEC, version 4.13.0) - blow by blower and Crank case

#### blowbyCyclic.st - Cyclic code
```iecst
(*******************************************************************************
AGGR: blowby			Blow by  (cyclic)

This code is confidential and proprietary to the INNIO Company.
It may not be used in any form, or reproduced in any manner, without the express
written permission of the INNIO Company.
Copyright, INNIO Company, 2023

Customized modifications: -
------------------------

History:
-------
V3.20.0			13.04.2010	koppm.		new
V3.59.0 		04.06.2014	Tinello 	new spezification
V4.00.0  		29.01.2015	Mari 		Porting J920 FOR XT4
				13.05.2015	lettenb.	release FOR error monitoring: bParaSetupOk added to avoid err.msg at plc startup
V4.00.1			25.06.2015	lettenb.	twice declared param.removed(bPr_CC_Exist,rP_CC_MonActive,rPr_CC_HiHi)
				22.07.2015				adaption for BR6
V4.03.0			02.10.2015	lettenb.	blowby filter pressure monitoring added	acc. spec.(CM&U)
V4.04.0			16.06.2016	Tinello.	Doppelte Anbindung W2653 entfernt
V4.05.0			08.05.2017	lettenb.	Para.bBbOp_EOP added (request holecek)
V4.05.1			21.02.2018				xTOF_EOP: NOT added, fan operation only with closed oil valve, bugfix
V4.10.0			11.11.2020	Schmid		blow-by blower off in full load operation
V4.11.0			02.02.2022	Schmid		suppress crankcase pressure max trip in case of load rejection or grid code event
V4.13.0			28.06.2023	Tinello		Blow-by fan needs to be operated when oil pump is running

Instructions for use:
--------------------

Outstandings:
------------

*******************************************************************************)
PROGRAM _CYCLIC

	(*----------------------------------*)
	(* RESET of alarms and warnings 	*)
	(*----------------------------------*)
	bAMM_BbBlower_Not_Rdy		:= FALSE;
	bAMM_Pc_BbBlower_Hi 		:= FALSE;

	bAMM_Pr_f_BbFilt_Ms			:= FALSE;
	bAMM_Pr_f_BbFilt_A_Ms		:= FALSE;
	bAMM_Pr_f_BbFilt_B_Ms		:= FALSE;
	bAMM_Pr_a_BbFilt_Ms			:= FALSE;
	bAMM_Pr_a_BbFilt_A_Ms		:= FALSE;
	bAMM_Pr_a_BbFilt_B_Ms		:= FALSE;

	bAMM_DPr_BbFilt_Hi			:= FALSE;
	bAMM_DPr_BbFilt_A_Hi		:= FALSE;
	bAMM_DPr_BbFilt_B_Hi		:= FALSE;
	bAMM_DPr_BbFilt_Lo			:= FALSE;
	bAMM_DPr_BbFilt_A_Lo		:= FALSE;
	bAMM_DPr_BbFilt_B_Lo		:= FALSE;
	bAMM_Pr_CC_MsMs				:= FALSE;
	bAMM_Pr_CC_Lo				:= FALSE;
	bAMM_Pr_CC_Hi				:= FALSE;
	bAMM_Pr_CC_HiHi				:= FALSE;

	(*----------------------------------*)
	(* Blow by blower				 	*)
	(*----------------------------------*)
	xTOF_EOP(IN:= OUT_AG.tEOP1AC_Dem.Do OR OUT_AG.tTC_EOP_On.Do, PT:= T#5m);

	xGR_MAXR_P_Act_Norm_Filt(In:= IN_AG.rP_Act_Norm_Filt, Gw:= Para.rP_Norm_BbBlower_off, Hy:= 0.02);
	xGR_MAXR_P_Set_Norm(In:= IN_AG.rP_Set_Norm, Gw:= Para.rP_Norm_BbBlower_off, Hy:= 0.02);
	xGR_MINR_Pr_CC(In:= IN_AG.tPr_CC.Ai, Gw:= -0.005, Hy:= 0.003);
	xTON_BbBlower_SS(IN:= xGR_MAXR_P_Act_Norm_Filt.Q AND xGR_MAXR_P_Set_Norm.Q AND xGR_MINR_Pr_CC.Q, PT:= T#10s);

	bBbBlower_Off := xTON_BbBlower_SS.Q AND IN_AG.bEng_Aux_Dem AND Para.bBbBlower_Off_Active;

	OUT_AG.tBbBlower.Do 		:=	(IN_AG.bEng_Aux_Dem_CDR OR (Para.bBbOp_EOP AND xTOF_EOP.Q))
								AND	NOT bBbBlower_Off;

	IF MM2VIS.bMsg3323 	THEN			(* crank case pressure - measurement signal failure *)
		OUT_AG.tBbBlower_y.Ao 	:= LIMIT(0, IN_AG.rP_Act_Norm_Filt, rPc_BbBlower_Save);	(* crank case controller output *)
	ELSE
		OUT_AG.tBbBlower_y.Ao 	:= rPc_BbBlower;
		rPc_BbBlower_Save		:= rPc_BbBlower;
	END_IF;

	(*--------------------------------------*)
	(* Blow by filter difference pressure	*)
	(*--------------------------------------*)
	(* Calculation of blow-by filter difference pressure *)
	rDPr_BbFilt		:= ABS(IN_AG.tPr_a_BbFilt.Ai   - IN_AG.tPr_f_BbFilt.Ai);
	rDPr_BbFilt_A	:= ABS(IN_AG.tPr_a_BbFilt_A.Ai - IN_AG.tPr_f_BbFilt_A.Ai);
	rDPr_BbFilt_B	:= ABS(IN_AG.tPr_a_BbFilt_B.Ai - IN_AG.tPr_f_BbFilt_B.Ai);

	(*--------------------------------------*)
	(* crank case pressure monitoring       *)
	(*--------------------------------------*)
	xTOF_BlocTrip_Pr_CC_HiHi.IN	:=	EDGEPOS(IN_AG.bLR_ActSat_CBV OR IN_AG.bGrC_HBErr_AUS); (* load rejection or grid code event *)
	xTOF_BlocTrip_Pr_CC_HiHi.PT	:=	T#30s;
	xTOF_BlocTrip_Pr_CC_HiHi();

	(*--------------------------------------------------*)
	(* release for error monitoring 					*)
	(*--------------------------------------------------*)
	IF bOMSS_MAT AND IN_AG.tPB2MM.bParaSetupOk THEN
		(*------------------------------------------------------------------*)
		(* measurement signal failure 										*)
		(*------------------------------------------------------------------*)
		bAMM_Pr_CC_MsMs 		:= Para.bPr_CC_MS_Exist	   		AND NOT IN_AG.tPr_CC.GoodQual; 			(* A3323 *)
		(* pressure before blow by filter *)
		bAMM_Pr_f_BbFilt_Ms		:= Para.bPr_f_BbFilt_Exist 		AND NOT IN_AG.tPr_f_BbFilt.GoodQual; 	(* W2651 *)
		bAMM_Pr_f_BbFilt_A_Ms	:= Para.bPr_f_BbFilt_A_Exist 	AND NOT IN_AG.tPr_f_BbFilt_A.GoodQual;	(* W2754 *)
		bAMM_Pr_f_BbFilt_B_Ms	:= Para.bPr_f_BbFilt_B_Exist 	AND NOT IN_AG.tPr_f_BbFilt_B.GoodQual;	(* W2755 *)
		(* pressure after blow by filter *)
		bAMM_Pr_a_BbFilt_Ms 	:= Para.bPr_a_BbFilt_Exist 		AND NOT IN_AG.tPr_a_BbFilt.GoodQual;	(* W2652 *)
		bAMM_Pr_a_BbFilt_A_Ms	:= Para.bPr_a_BbFilt_A_Exist 	AND NOT IN_AG.tPr_a_BbFilt_A.GoodQual;	(* W2756 *)
		bAMM_Pr_a_BbFilt_B_Ms	:= Para.bPr_a_BbFilt_B_Exist 	AND NOT IN_AG.tPr_a_BbFilt_B.GoodQual;	(* W2757 *)

		(* Release monitoring	*)
		xTOF_AMM_Pr_CC_MsMs      (IN:= bAMM_Pr_CC_MsMs, 	  PT:= T#10s);
		xTOF_AMM_Pr_f_BbFilt_Ms  (IN:= bAMM_Pr_f_BbFilt_Ms,   PT:= T#10s);	(* TOF because of filtered signals *)
		xTOF_AMM_Pr_f_BbFilt_A_Ms(IN:= bAMM_Pr_f_BbFilt_A_Ms, PT:= T#10s);
		xTOF_AMM_Pr_f_BbFilt_B_Ms(IN:= bAMM_Pr_f_BbFilt_B_Ms, PT:= T#10s);
		xTOF_AMM_Pr_a_BbFilt_Ms  (IN:= bAMM_Pr_a_BbFilt_Ms,   PT:= T#10s);
		xTOF_AMM_Pr_a_BbFilt_A_Ms(IN:= bAMM_Pr_a_BbFilt_A_Ms, PT:= T#10s);
		xTOF_AMM_Pr_a_BbFilt_B_Ms(IN:= bAMM_Pr_a_BbFilt_B_Ms, PT:= T#10s);

		bRelMon_Pr_CC			:= Para.bPr_CC_MS_Exist			AND NOT xTOF_AMM_Pr_CC_MsMs.Q;
		bRelMon_Pr_f_BbFilt		:= Para.bPr_f_BbFilt_Exist 		AND NOT xTOF_AMM_Pr_f_BbFilt_Ms.Q;
		bRelMon_Pr_f_BbFilt_A	:= Para.bPr_f_BbFilt_A_Exist 	AND NOT xTOF_AMM_Pr_f_BbFilt_A_Ms.Q;
		bRelMon_Pr_f_BbFilt_B	:= Para.bPr_f_BbFilt_B_Exist 	AND NOT xTOF_AMM_Pr_f_BbFilt_B_Ms.Q;
		bRelMon_Pr_a_BbFilt		:= Para.bPr_a_BbFilt_Exist 		AND NOT xTOF_AMM_Pr_a_BbFilt_Ms.Q;
		bRelMon_Pr_a_BbFilt_A	:= Para.bPr_a_BbFilt_A_Exist 	AND NOT xTOF_AMM_Pr_a_BbFilt_A_Ms.Q;
		bRelMon_Pr_a_BbFilt_B	:= Para.bPr_a_BbFilt_B_Exist 	AND NOT xTOF_AMM_Pr_a_BbFilt_B_Ms.Q;

		(*------------------------------------------------------------------*)
		(* monitoring blow-by filter difference pressure 					*)
		(*------------------------------------------------------------------*)
		IF 	(IN_AG.rP_Act_Norm_Filt > Para.rDPr_BbFilt_Pstart) 	AND		(* monitoring according to actual power *)
			IN_AG.bEng_Aux_Dem_CDR										(* engine is running *)
		THEN
			(* interpolation of MAXIMAL tolerated blow-by filter difference pressure *)
			xSigScal_R_DPrHi.X	:= IN_AG.rP_Act_Norm_Filt;
			xSigScal_R_DPrHi.X1 := Para.rDPr_BbFilt_Pstart;
			xSigScal_R_DPrHi.Y1 := Para.rDPr_BbFilt_Hi_P1;
			xSigScal_R_DPrHi.X2 := 1.0; 						(* 100% = nominal power *)
			xSigScal_R_DPrHi.Y2 := Para.rDPr_BbFilt_Hi_P2;
			xSigScal_R_DPrHi();

			(* interpolation of MINIMAL tolerated blow-by filter difference pressure *)
			xSigScal_R_DPrLo.X	:= IN_AG.rP_Act_Norm_Filt;
			xSigScal_R_DPrLo.X1 := Para.rDPr_BbFilt_Pstart;
			xSigScal_R_DPrLo.Y1 := Para.rDPr_BbFilt_Lo_P1;
			xSigScal_R_DPrLo.X2 := 1.0; 						(* 100% = nominal power *)
			xSigScal_R_DPrLo.Y2 := Para.rDPr_BbFilt_Lo_P2;
			xSigScal_R_DPrLo();

			IF (bRelMon_Pr_a_BbFilt AND bRelMon_Pr_f_BbFilt) THEN
				bAMM_DPr_BbFilt_Hi		:= (rDPr_BbFilt   >  xSigScal_R_DPrHi.Y_SCAL);									(* W2653 *)
				bAMM_DPr_BbFilt_Lo		:= (rDPr_BbFilt   < (xSigScal_R_DPrLo.Y_SCAL * 0.75));							(* W2654 *)
			END_IF;

			IF (bRelMon_Pr_a_BbFilt_A AND bRelMon_Pr_f_BbFilt_A) THEN
				bAMM_DPr_BbFilt_A_Hi	:= (rDPr_BbFilt_A >  xSigScal_R_DPrHi.Y_SCAL);									(* W2758 *)
				bAMM_DPr_BbFilt_A_Lo	:= (rDPr_BbFilt_A < (xSigScal_R_DPrLo.Y_SCAL * 0.75));							(* W2760 *)
			END_IF;

			IF (bRelMon_Pr_a_BbFilt_B AND bRelMon_Pr_f_BbFilt_B) THEN
				bAMM_DPr_BbFilt_B_Hi	:= (rDPr_BbFilt_B >  xSigScal_R_DPrHi.Y_SCAL);									(* W2759 *)
				bAMM_DPr_BbFilt_B_Lo	:= (rDPr_BbFilt_B < (xSigScal_R_DPrLo.Y_SCAL * 0.75));							(* W2761 *)
			END_IF;
		END_IF;

		(*------------------------------------------------------------------*)
		(* Blow by blower			 										*)
		(*------------------------------------------------------------------*)
		(* error by DI *)
		bAMM_BbBlower_Not_Rdy	:= NOT IN_AG.tBbBlower_FC_Rdy.Di; 			(* M.03-M-001 *)							(* W2650 *)

		(* error blow by blower SPEED max *)
		bAMM_Pc_BbBlower_Hi 	:= (rPc_BbBlower > Para.rPc_BbBlower_Hi) AND OUT_AG.tBbBlower.Do AND Para.bCtr_CC;		(* W2591 *)

		(*----------------------------------------------------------------------*)
		(* monitoring crank case pressure according to actual power				*)
		(*----------------------------------------------------------------------*)
		IF 	bRelMon_Pr_CC AND (IN_AG.rP_Act_Norm_Filt > Para.rP_CC_MonActive_LimHi)
		THEN
			(*--------------------------------------------------*)
			(* crank case pressure MIN 					  		*)
			(*--------------------------------------------------*)
			bAMM_Pr_CC_Lo 		:= IN_AG.tPr_CC.Ai < Para.rPr_CC_Lo;													(* W2649 *)

			(*--------------------------------------------------*)
			(* crank case pressure MAX / POWER REDUCTION  		*)
			(*--------------------------------------------------*)
			bAMM_Pr_CC_Hi 		:= IN_AG.tPr_CC.Ai > Para.rPr_CC_Hi;													(* W2558 *)

			IF xEngType.Type9 THEN
				(* power reduction from actual power step by step *)													(* B2875 *)
				xTON_Pr_CC_Hi(IN:= (IN_AG.tPr_CC.Ai >= Para.rPr_CC_Hi) AND NOT xTON_Pr_CC_Hi.Q, PT:= Para.tiPr_CC_Hi);

				IF xTON_Pr_CC_Hi.Q THEN
					OUT_AG.rP_Red_Pr_CC_Norm 	:= LIMIT(0, rP_Act_Norm_Save - Para.rP_Red_CC, 1.0);
				ELSE
					rP_Act_Norm_Save			:= IN_AG.rP_Act_Norm_Filt;		(* save actual power *)
				END_IF;

				(* Reset power reduction step by step *)
				xTON_Pr_CC_OK(IN:= (IN_AG.tPr_CC.Ai < Para.rPr_CC_Hi) AND (OUT_AG.rP_Red_Pr_CC_Norm < 1.0) AND NOT xTON_Pr_CC_OK.Q,
							  PT:= T#60s);

				IF xTON_Pr_CC_OK.Q THEN
					OUT_AG.rP_Red_Pr_CC_Norm	:= LIMIT(0, OUT_AG.rP_Red_Pr_CC_Norm + Para.rP_Red_CC, 1.0);
				END_IF;
			ELSE
				(* Reset power reduction *)
				xTON_Pr_CC_Hi(IN:= FALSE);
				xTON_Pr_CC_OK(IN:= FALSE);
				OUT_AG.rP_Red_Pr_CC_Norm 		:= 1.0;			(* release full load - no reduction *)
			END_IF;

			(*--------------------------------------------------*)
			(* crank case pressure MAX / SHUT DOWN		  		*)
			(*--------------------------------------------------*)
			xTON_Pr_CC_HiHi(IN	:= IN_AG.tPr_CC.Ai > Para.rPr_CC_LimHiHi, PT:= Para.tiPr_CC_HiHi);
			bAMM_Pr_CC_HiHi 	:= xTON_Pr_CC_HiHi.Q AND NOT xTOF_BlocTrip_Pr_CC_HiHi.Q;								(* A3322 *)
		ELSE
			(* Reset power reduction *)
			xTON_Pr_CC_Hi	(IN:= FALSE);
			xTON_Pr_CC_OK	(IN:= FALSE);
			xTON_Pr_CC_HiHi	(IN:= FALSE);
			OUT_AG.rP_Red_Pr_CC_Norm 		:= 1.0;			(* release full load - no reduction *)
		END_IF;

		(*----------------------------------------------------------------------*)
		(* monitoring crank case pressure independent to actual power			*)
		(*----------------------------------------------------------------------*)
		(*--------------------------------------------------*)
		(* crank case pressure MAX / SHUT DOWN		  		*)
		(*--------------------------------------------------*)
		bAMM_Pr_CC_HiHi 	:=	((IN_AG.tPr_CC.Ai > (Para.rPr_CC_LimHiHi + 0.002) AND bRelMon_Pr_CC) OR bAMM_Pr_CC_HiHi)	(* A3322 *)
							AND	NOT xTOF_BlocTrip_Pr_CC_HiHi.Q;

	ELSE
		(* Reset monitoring TOF	*)
		xTOF_AMM_Pr_CC_MsMs      (IN:= FALSE, PT:= T#0s);
		xTOF_AMM_Pr_f_BbFilt_Ms  (IN:= FALSE, PT:= T#0s);
		xTOF_AMM_Pr_f_BbFilt_A_Ms(IN:= FALSE, PT:= T#0s);
		xTOF_AMM_Pr_f_BbFilt_B_Ms(IN:= FALSE, PT:= T#0s);
		xTOF_AMM_Pr_a_BbFilt_Ms  (IN:= FALSE, PT:= T#0s);
		xTOF_AMM_Pr_a_BbFilt_A_Ms(IN:= FALSE, PT:= T#0s);
		xTOF_AMM_Pr_a_BbFilt_B_Ms(IN:= FALSE, PT:= T#0s);

		(* Reset power reduction *)
		xTON_Pr_CC_Hi	(IN:= FALSE);
		xTON_Pr_CC_OK	(IN:= FALSE);
		xTON_Pr_CC_HiHi	(IN:= FALSE);
		OUT_AG.rP_Red_Pr_CC_Norm	:= 1.0;					(* release full load - no reduction *)
	END_IF;

END_PROGRAM
```

#### blowby.var - Local variables
```iecst
VAR
	bRelMon_Pr_CC : BOOL := FALSE; (*Release monitoring crank case pressure*)
	bRelMon_Pr_a_BbFilt : BOOL := FALSE; (*Release monitoring pressure after blow by filter *)
	bRelMon_Pr_f_BbFilt : BOOL := FALSE; (*Release monitoring pressure before blow by filter *)
	bRelMon_Pr_a_BbFilt_A : BOOL := FALSE; (*Release monitoring pressure after blow by filter Bank A*)
	bRelMon_Pr_a_BbFilt_B : BOOL := FALSE; (*Release monitoring pressure after blow by filter Bank B*)
	bRelMon_Pr_f_BbFilt_A : BOOL := FALSE; (*Release monitoring pressure before blow by filter Bank A*)
	bRelMon_Pr_f_BbFilt_B : BOOL := FALSE; (*Release monitoring pressure before blow by filter Bank B*)

	rPc_BbBlower_Save : REAL := 0; (*Saved controller output before error [%]*)
	rP_Act_Norm_Save : REAL := 0.0; (*SAVE actual power related to rP_Nom [% Pnom] filtered T=1s*)
	xSigScal_R_DPrHi : xSigScal_R := (0);
	xSigScal_R_DPrLo : xSigScal_R := (0);

	xTOF_AMM_Pr_CC_MsMs : TOF := (0);
	xTOF_AMM_Pr_a_BbFilt_Ms : TOF := (0);
	xTOF_AMM_Pr_a_BbFilt_A_Ms : TOF := (0);
	xTOF_AMM_Pr_a_BbFilt_B_Ms : TOF := (0);
	xTOF_AMM_Pr_f_BbFilt_Ms : TOF := (0);
	xTOF_AMM_Pr_f_BbFilt_A_Ms : TOF := (0);
	xTOF_AMM_Pr_f_BbFilt_B_Ms : TOF := (0);

	xTON_Pr_CC_Hi : TON := (0);
	xTON_Pr_CC_HiHi : TON := (0);
	xTON_Pr_CC_OK : TON := (0);
	xTOF_BlocTrip_Pr_CC_HiHi : TOF;

	xTOF_EOP : TOF := (0);

	xGR_MAXR_P_Act_Norm_Filt : GR_MAXR;
	xGR_MINR_Pr_CC : GR_MINR;
	xGR_MAXR_P_Set_Norm : GR_MAXR;
	xTON_BbBlower_SS : TON;
	bBbBlower_Off : BOOL;
END_VAR
```

### Program Logical/AuxiliariesGeneral/Ctr_CC (IEC, version 4.11.0) - controller crank case pressure
